Yaskawa INFORM job: A_ROOF_SIDE_0617_2_PAINT_11.JBI

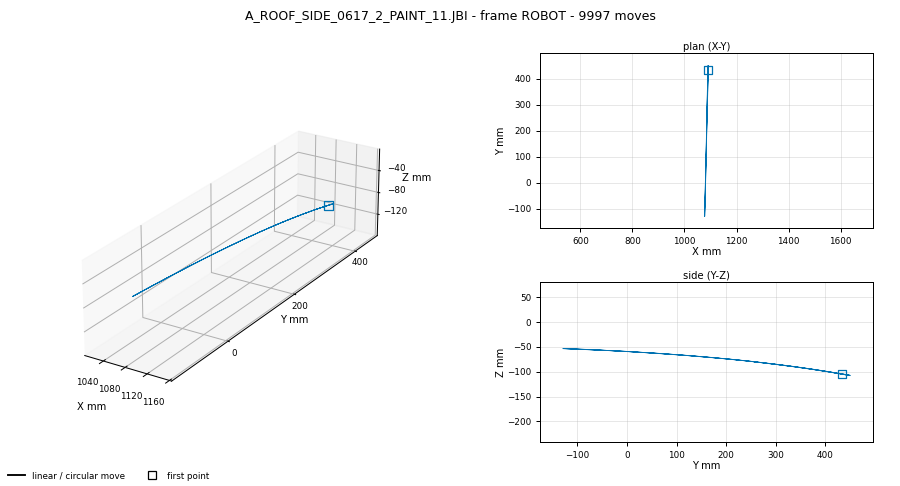
[picture p0: tool path of A_ROOF_SIDE_0617_2_PAINT_11.JBI in frame ROBOT, 9997 of 9997 moves have a stored position in this frame; points joined in program order, loops and branches not executed]
/JOB
//NAME A_ROOF_SIDE_0617_2_PAINT11
//POS
///NPOS 9997,0,0,0,0,0
///TOOL 1
///USER 0
///POSTYPE ROBOT
///RECTAN
///RCONF 1,0,0,0,0,0,0,0,0,0,0,0,0,0,0,0,0,0,0,0,0,0,0,0
C00000=1091.867,433.561,-104.062,178.470,26.056,154.096
C00001=1091.874,433.807,-104.105,178.473,26.068,154.099
C00002=1091.880,434.053,-104.148,178.477,26.080,154.102
C00003=1091.887,434.299,-104.192,178.480,26.092,154.104
C00004=1091.893,434.545,-104.234,178.484,26.104,154.107
C00005=1091.899,434.791,-104.277,178.486,26.116,154.110
C00006=1091.906,435.037,-104.321,178.490,26.128,154.112
C00007=1091.912,435.283,-104.365,178.493,26.141,154.115
C00008=1091.918,435.530,-104.408,178.497,26.153,154.117
C00009=1091.926,435.775,-104.451,178.500,26.165,154.120
C00010=1091.932,436.022,-104.494,178.503,26.177,154.123
C00011=1091.938,436.268,-104.538,178.507,26.189,154.126
C00012=1091.945,436.514,-104.581,178.510,26.202,154.128
C00013=1091.951,436.760,-104.624,178.513,26.214,154.131
C00014=1091.958,437.006,-104.668,178.517,26.227,154.134
C00015=1091.965,437.252,-104.711,178.520,26.239,154.137
C00016=1091.971,437.498,-104.755,178.524,26.252,154.139
C00017=1091.978,437.744,-104.799,178.527,26.264,154.142
C00018=1091.988,438.137,-104.869,178.533,26.285,154.147
C00019=1091.999,438.531,-104.938,178.538,26.305,154.151
C00020=1092.009,438.925,-105.008,178.543,26.326,154.156
C00021=1092.020,439.319,-105.078,178.548,26.346,154.160
C00022=1092.027,439.565,-105.122,178.552,26.359,154.163
C00023=1092.033,439.811,-105.166,178.556,26.372,154.166
C00024=1092.041,440.056,-105.210,178.559,26.385,154.169
C00025=1092.047,440.302,-105.254,178.562,26.398,154.172
C00026=1092.053,440.548,-105.297,178.565,26.411,154.175
C00027=1092.060,440.794,-105.341,178.569,26.424,154.178
C00028=1092.067,441.041,-105.385,178.572,26.438,154.181
C00029=1092.074,441.286,-105.430,178.575,26.451,154.184
C00030=1092.080,441.532,-105.474,178.579,26.464,154.187
C00031=1092.086,441.778,-105.518,178.583,26.478,154.190
C00032=1092.093,442.023,-105.562,178.586,26.491,154.193
C00033=1092.100,442.269,-105.606,178.589,26.504,154.196
C00034=1092.107,442.516,-105.650,178.593,26.518,154.199
C00035=1092.113,442.761,-105.695,178.596,26.532,154.202
C00036=1092.120,443.007,-105.739,178.600,26.546,154.205
C00037=1092.127,443.253,-105.783,178.603,26.559,154.208
C00038=1092.132,443.499,-105.828,178.606,26.573,154.211
C00039=1092.140,443.745,-105.873,178.610,26.586,154.214
C00040=1092.146,443.991,-105.917,178.614,26.601,154.218
C00041=1092.153,444.236,-105.961,178.616,26.614,154.221
C00042=1092.159,444.482,-106.006,178.620,26.628,154.224
C00043=1092.166,444.728,-106.050,178.624,26.642,154.227
C00044=1092.173,444.974,-106.094,178.626,26.656,154.230
C00045=1092.180,445.220,-106.140,178.629,26.670,154.233
C00046=1092.186,445.466,-106.185,178.632,26.684,154.237
C00047=1092.193,445.711,-106.228,178.633,26.697,154.240
C00048=1092.200,445.958,-106.273,178.636,26.711,154.243
C00049=1092.206,446.203,-106.318,178.638,26.725,154.246
C00050=1092.213,446.449,-106.363,178.639,26.739,154.250
C00051=1092.220,446.695,-106.408,178.641,26.752,154.253
C00052=1092.227,446.940,-106.453,178.643,26.767,154.256
C00053=1092.233,447.186,-106.498,178.644,26.780,154.260
C00054=1092.240,447.432,-106.543,178.645,26.794,154.263
C00055=1092.246,447.677,-106.588,178.646,26.807,154.267
C00056=1092.254,447.923,-106.633,178.647,26.821,154.270
C00057=1092.260,448.169,-106.677,178.648,26.835,154.273
C00058=1092.267,448.415,-106.723,178.648,26.849,154.277
C00059=1092.274,448.660,-106.767,178.649,26.862,154.280
C00060=1092.281,448.907,-106.812,178.649,26.876,154.284
C00061=1092.287,449.152,-106.857,178.650,26.890,154.287
C00062=1092.294,449.398,-106.902,178.649,26.903,154.291
C00063=1092.301,449.644,-106.947,178.649,26.917,154.294
C00064=1092.308,449.888,-106.992,178.649,26.931,154.298
C00065=1092.317,450.135,-107.036,178.649,26.943,154.301
C00066=1091.932,450.127,-107.217,178.601,27.145,154.357
C00067=1091.923,449.881,-107.173,178.601,27.132,154.354
C00068=1091.915,449.636,-107.127,178.601,27.119,154.350
C00069=1091.908,449.390,-107.082,178.601,27.105,154.347
C00070=1091.902,449.145,-107.037,178.601,27.091,154.343
C00071=1091.895,448.899,-106.992,178.601,27.078,154.340
C00072=1091.888,448.654,-106.947,178.601,27.064,154.336
C00073=1091.881,448.407,-106.902,178.600,27.050,154.333
C00074=1091.875,448.162,-106.857,178.600,27.037,154.330
C00075=1091.868,447.916,-106.811,178.599,27.023,154.326
C00076=1091.861,447.670,-106.767,178.598,27.009,154.323
C00077=1091.854,447.424,-106.722,178.596,26.995,154.319
C00078=1091.848,447.179,-106.677,178.595,26.982,154.316
C00079=1091.841,446.933,-106.632,178.594,26.968,154.313
C00080=1091.834,446.687,-106.587,178.592,26.954,154.309
C00081=1091.827,446.441,-106.542,178.591,26.940,154.306
C00082=1091.821,446.196,-106.497,178.588,26.926,154.303
C00083=1091.814,445.950,-106.453,178.586,26.912,154.299
C00084=1091.807,445.704,-106.407,178.585,26.898,154.296
C00085=1091.800,445.458,-106.363,178.582,26.884,154.293
C00086=1091.793,445.212,-106.318,178.579,26.871,154.290
C00087=1091.787,444.966,-106.274,178.576,26.857,154.286
C00088=1091.780,444.721,-106.229,178.573,26.843,154.283
C00089=1091.773,444.475,-106.184,178.570,26.829,154.280
C00090=1091.767,444.229,-106.139,178.567,26.815,154.277
C00091=1091.760,443.983,-106.095,178.563,26.801,154.274
C00092=1091.753,443.737,-106.050,178.559,26.787,154.270
C00093=1091.746,443.492,-106.006,178.556,26.773,154.267
C00094=1091.740,443.246,-105.962,178.553,26.760,154.264
C00095=1091.733,443.001,-105.917,178.549,26.746,154.261
C00096=1091.727,442.754,-105.873,178.545,26.732,154.258
C00097=1091.720,442.508,-105.828,178.542,26.718,154.255
C00098=1091.714,442.262,-105.784,178.539,26.705,154.252
C00099=1091.707,442.017,-105.740,178.535,26.691,154.249
C00100=1091.700,441.770,-105.695,178.531,26.678,154.246
C00101=1091.693,441.525,-105.651,178.527,26.664,154.243
C00102=1091.687,441.279,-105.607,178.525,26.651,154.240
C00103=1091.680,441.033,-105.563,178.521,26.637,154.237
C00104=1091.674,440.788,-105.519,178.517,26.624,154.234
C00105=1091.667,440.542,-105.475,178.514,26.611,154.231
C00106=1091.660,440.296,-105.431,178.510,26.598,154.228
C00107=1091.653,440.049,-105.387,178.508,26.585,154.225
C00108=1091.646,439.804,-105.343,178.504,26.572,154.222
C00109=1091.640,439.558,-105.299,178.500,26.559,154.219
C00110=1091.633,439.312,-105.255,178.497,26.546,154.216
C00111=1091.622,438.929,-105.187,178.491,26.526,154.212
C00112=1091.612,438.547,-105.119,178.486,26.506,154.207
C00113=1091.602,438.165,-105.050,178.481,26.486,154.203
C00114=1091.592,437.783,-104.983,178.475,26.466,154.198
C00115=1091.585,437.537,-104.939,178.471,26.454,154.196
C00116=1091.579,437.291,-104.896,178.469,26.441,154.193
C00117=1091.572,437.045,-104.853,178.465,26.428,154.190
C00118=1091.566,436.799,-104.809,178.462,26.416,154.187
C00119=1091.559,436.553,-104.765,178.458,26.403,154.185
C00120=1091.552,436.307,-104.722,178.455,26.391,154.182
C00121=1091.546,436.061,-104.678,178.451,26.378,154.179
C00122=1091.540,435.815,-104.635,178.448,26.367,154.176
C00123=1091.532,435.569,-104.591,178.444,26.354,154.174
C00124=1091.526,435.322,-104.548,178.441,26.342,154.171
C00125=1091.520,435.076,-104.504,178.437,26.329,154.168
C00126=1091.513,434.831,-104.461,178.434,26.317,154.166
C00127=1091.507,434.584,-104.418,178.431,26.305,154.163
C00128=1091.500,434.338,-104.374,178.427,26.293,154.160
C00129=1091.493,434.092,-104.332,178.424,26.281,154.158
C00130=1091.487,433.846,-104.288,178.420,26.268,154.155
C00131=1091.481,433.600,-104.246,178.417,26.257,154.152
C00132=1091.474,433.354,-104.202,178.414,26.245,154.150
C00133=1091.468,433.108,-104.159,178.410,26.233,154.147
C00134=1091.461,432.861,-104.116,178.407,26.221,154.144
C00135=1091.455,432.615,-104.072,178.403,26.209,154.142
C00136=1091.448,432.369,-104.030,178.400,26.197,154.139
C00137=1091.441,432.123,-103.987,178.397,26.186,154.137
C00138=1091.436,431.877,-103.944,178.393,26.174,154.134
C00139=1091.428,431.631,-103.901,178.390,26.162,154.132
C00140=1091.422,431.385,-103.858,178.387,26.151,154.129
C00141=1091.415,431.138,-103.815,178.383,26.139,154.127
C00142=1091.409,430.892,-103.773,178.380,26.128,154.124
C00143=1091.403,430.646,-103.730,178.377,26.117,154.122
C00144=1091.396,430.400,-103.688,178.374,26.105,154.119
C00145=1091.389,430.154,-103.645,178.370,26.094,154.117
C00146=1091.383,429.907,-103.602,178.367,26.082,154.114
C00147=1091.377,429.662,-103.560,178.364,26.071,154.112
C00148=1091.370,429.415,-103.517,178.360,26.060,154.110
C00149=1091.364,429.169,-103.474,178.356,26.048,154.107
C00150=1091.358,428.923,-103.432,178.353,26.037,154.105
C00151=1091.351,428.677,-103.389,178.350,26.026,154.102
C00152=1091.345,428.430,-103.346,178.347,26.015,154.100
C00153=1091.338,428.184,-103.304,178.343,26.004,154.097
C00154=1091.332,427.938,-103.261,178.340,25.993,154.095
C00155=1091.325,427.691,-103.220,178.337,25.982,154.093
C00156=1091.318,427.445,-103.177,178.333,25.971,154.090
C00157=1091.312,427.200,-103.135,178.330,25.960,154.088
C00158=1091.305,426.953,-103.092,178.326,25.949,154.086
C00159=1091.299,426.706,-103.050,178.323,25.938,154.083
C00160=1091.293,426.460,-103.008,178.320,25.927,154.081
C00161=1091.287,426.214,-102.966,178.317,25.916,154.079
C00162=1091.280,425.967,-102.923,178.313,25.906,154.077
C00163=1091.273,425.736,-102.884,178.310,25.895,154.074
C00164=1091.268,425.503,-102.844,178.307,25.885,154.072
C00165=1091.261,425.271,-102.804,178.304,25.876,154.070
C00166=1091.256,425.039,-102.765,178.301,25.866,154.068
C00167=1091.249,424.807,-102.725,178.298,25.856,154.066
C00168=1091.244,424.574,-102.686,178.294,25.846,154.064
C00169=1091.238,424.343,-102.646,178.292,25.836,154.062
C00170=1091.231,424.110,-102.607,178.288,25.826,154.060
C00171=1091.225,423.864,-102.565,178.285,25.815,154.057
C00172=1091.218,423.618,-102.523,178.282,25.805,154.055
C00173=1091.213,423.371,-102.481,178.279,25.794,154.053
C00174=1091.206,423.124,-102.440,178.275,25.784,154.051
C00175=1091.200,422.879,-102.397,178.272,25.774,154.049
C00176=1091.193,422.632,-102.356,178.269,25.764,154.046
C00177=1091.187,422.386,-102.314,178.266,25.753,154.044
C00178=1091.181,422.139,-102.272,178.262,25.743,154.042
C00179=1091.175,421.893,-102.231,178.259,25.733,154.040
C00180=1091.168,421.646,-102.188,178.256,25.723,154.038
C00181=1091.162,421.400,-102.147,178.252,25.713,154.036
C00182=1091.155,421.154,-102.106,178.249,25.703,154.034
C00183=1091.149,420.907,-102.064,178.246,25.693,154.032
C00184=1091.142,420.660,-102.022,178.243,25.682,154.029
C00185=1091.136,420.414,-101.981,178.239,25.672,154.027
C00186=1091.130,420.168,-101.939,178.236,25.662,154.025
C00187=1091.123,419.921,-101.898,178.233,25.653,154.023
C00188=1091.117,419.675,-101.857,178.229,25.642,154.021
C00189=1091.110,419.428,-101.815,178.226,25.633,154.019
C00190=1091.105,419.182,-101.773,178.223,25.623,154.017
C00191=1091.098,418.936,-101.733,178.219,25.613,154.015
C00192=1091.092,418.689,-101.691,178.217,25.603,154.013
C00193=1091.086,418.442,-101.650,178.214,25.594,154.011
C00194=1091.079,418.197,-101.609,178.210,25.584,154.009
C00195=1091.072,417.950,-101.567,178.207,25.574,154.007
C00196=1091.067,417.703,-101.527,178.204,25.564,154.005
C00197=1091.061,417.457,-101.485,178.200,25.555,154.003
C00198=1091.054,417.210,-101.444,178.197,25.545,154.001
C00199=1091.048,416.963,-101.403,178.194,25.536,153.999
C00200=1091.042,416.717,-101.362,178.191,25.526,153.997
C00201=1091.035,416.471,-101.321,178.187,25.517,153.995
C00202=1091.029,416.224,-101.280,178.184,25.507,153.993
C00203=1091.022,415.978,-101.239,178.181,25.497,153.991
C00204=1091.017,415.731,-101.198,178.177,25.488,153.989
C00205=1091.009,415.484,-101.157,178.175,25.479,153.987
C00206=1091.004,415.237,-101.116,178.171,25.470,153.985
C00207=1090.997,414.992,-101.075,178.168,25.461,153.984
C00208=1090.991,414.744,-101.034,178.165,25.451,153.982
C00209=1090.984,414.498,-100.994,178.162,25.442,153.980
C00210=1090.978,414.252,-100.953,178.159,25.433,153.978
C00211=1090.972,414.005,-100.912,178.155,25.424,153.976
C00212=1090.965,413.759,-100.872,178.152,25.414,153.974
C00213=1090.959,413.511,-100.830,178.149,25.405,153.972
C00214=1090.953,413.265,-100.790,178.146,25.396,153.970
C00215=1090.946,413.018,-100.750,178.142,25.387,153.969
C00216=1090.940,412.772,-100.709,178.140,25.378,153.967
C00217=1090.934,412.526,-100.669,178.136,25.369,153.965
C00218=1090.928,412.278,-100.627,178.133,25.360,153.963
C00219=1090.922,412.054,-100.591,178.130,25.352,153.961
C00220=1090.917,411.829,-100.554,178.127,25.344,153.960
C00221=1090.911,411.605,-100.517,178.124,25.336,153.958
C00222=1090.905,411.380,-100.480,178.122,25.328,153.957
C00223=1090.899,411.155,-100.443,178.119,25.319,153.955
C00224=1090.894,410.930,-100.406,178.115,25.311,153.953
C00225=1090.887,410.706,-100.370,178.112,25.303,153.952
C00226=1090.882,410.481,-100.333,178.110,25.295,153.950
C00227=1090.876,410.234,-100.293,178.107,25.287,153.948
C00228=1090.870,409.987,-100.252,178.103,25.278,153.947
C00229=1090.864,409.741,-100.212,178.100,25.269,153.945
C00230=1090.857,409.494,-100.171,178.097,25.260,153.943
C00231=1090.852,409.247,-100.131,178.094,25.252,153.941
C00232=1090.845,409.001,-100.091,178.091,25.243,153.939
C00233=1090.839,408.754,-100.051,178.088,25.234,153.938
C00234=1090.833,408.507,-100.011,178.084,25.226,153.936
C00235=1090.827,408.260,-99.970,178.082,25.217,153.934
C00236=1090.821,408.014,-99.930,178.078,25.208,153.933
C00237=1090.814,407.767,-99.890,178.075,25.200,153.931
C00238=1090.808,407.520,-99.851,178.072,25.192,153.929
C00239=1090.802,407.274,-99.810,178.069,25.183,153.927
C00240=1090.795,407.027,-99.770,178.065,25.175,153.926
C00241=1090.790,406.780,-99.729,178.063,25.166,153.924
C00242=1090.784,406.533,-99.690,178.059,25.158,153.923
C00243=1090.777,406.287,-99.650,178.057,25.149,153.921
C00244=1090.772,406.041,-99.610,178.053,25.141,153.919
C00245=1090.766,405.794,-99.571,178.050,25.133,153.918
C00246=1090.759,405.547,-99.531,178.047,25.124,153.916
C00247=1090.753,405.300,-99.491,178.044,25.116,153.914
C00248=1090.747,405.054,-99.451,178.040,25.108,153.913
C00249=1090.741,404.806,-99.412,178.038,25.100,153.911
C00250=1090.734,404.560,-99.371,178.035,25.092,153.909
C00251=1090.728,404.313,-99.332,178.031,25.084,153.908
C00252=1090.722,404.066,-99.292,178.029,25.076,153.906
C00253=1090.716,403.819,-99.252,178.025,25.067,153.905
C00254=1090.710,403.573,-99.213,178.022,25.059,153.903
C00255=1090.703,403.326,-99.174,178.018,25.051,153.902
C00256=1090.697,403.079,-99.134,178.016,25.043,153.900
C00257=1090.691,402.833,-99.094,178.013,25.035,153.898
C00258=1090.685,402.586,-99.055,178.009,25.027,153.897
C00259=1090.679,402.339,-99.015,178.007,25.019,153.895
C00260=1090.672,402.091,-98.976,178.004,25.011,153.894
C00261=1090.667,401.846,-98.936,178.000,25.003,153.892
C00262=1090.660,401.599,-98.897,177.997,24.996,153.891
C00263=1090.654,401.352,-98.858,177.994,24.988,153.889
C00264=1090.648,401.105,-98.818,177.991,24.980,153.888
C00265=1090.642,400.859,-98.779,177.988,24.972,153.886
C00266=1090.636,400.612,-98.739,177.984,24.964,153.885
C00267=1090.629,400.365,-98.700,177.982,24.956,153.883
C00268=1090.623,400.118,-98.661,177.979,24.949,153.882
C00269=1090.617,399.871,-98.622,177.975,24.941,153.880
C00270=1090.611,399.624,-98.582,177.972,24.933,153.878
C00271=1090.605,399.377,-98.543,177.970,24.925,153.877
C00272=1090.599,399.130,-98.504,177.967,24.918,153.876
C00273=1090.593,398.884,-98.465,177.963,24.910,153.874
C00274=1090.586,398.637,-98.426,177.960,24.903,153.873
C00275=1090.581,398.413,-98.390,177.957,24.896,153.871
C00276=1090.575,398.188,-98.355,177.954,24.889,153.870
C00277=1090.570,397.964,-98.320,177.952,24.882,153.869
C00278=1090.564,397.740,-98.283,177.949,24.875,153.867
C00279=1090.558,397.515,-98.249,177.946,24.868,153.866
C00280=1090.553,397.291,-98.213,177.943,24.862,153.865
C00281=1090.547,397.067,-98.177,177.941,24.855,153.863
C00282=1090.543,396.843,-98.142,177.938,24.848,153.862
C00283=1090.536,396.596,-98.103,177.935,24.841,153.861
C00284=1090.530,396.349,-98.064,177.931,24.833,153.859
C00285=1090.524,396.102,-98.026,177.929,24.826,153.858
C00286=1090.518,395.855,-97.987,177.926,24.818,153.857
C00287=1090.512,395.609,-97.948,177.923,24.811,153.855
C00288=1090.506,395.361,-97.910,177.919,24.803,153.854
C00289=1090.500,395.114,-97.870,177.916,24.796,153.852
C00290=1090.493,394.868,-97.832,177.913,24.789,153.851
C00291=1090.487,394.621,-97.793,177.910,24.782,153.850
C00292=1090.481,394.374,-97.755,177.907,24.774,153.848
C00293=1090.475,394.127,-97.716,177.904,24.767,153.847
C00294=1090.469,393.880,-97.677,177.901,24.760,153.846
C00295=1090.463,393.633,-97.639,177.898,24.753,153.844
C00296=1090.457,393.387,-97.601,177.895,24.746,153.843
C00297=1090.451,393.140,-97.561,177.892,24.738,153.841
C00298=1090.444,392.893,-97.523,177.889,24.731,153.840
C00299=1090.439,392.646,-97.484,177.885,24.724,153.839
C00300=1090.433,392.400,-97.446,177.882,24.717,153.838
C00301=1090.426,392.152,-97.408,177.879,24.710,153.836
C00302=1090.421,391.905,-97.369,177.876,24.703,153.835
C00303=1090.414,391.658,-97.330,177.873,24.696,153.834
C00304=1090.408,391.412,-97.293,177.870,24.689,153.832
C00305=1090.401,391.165,-97.254,177.866,24.682,153.831
C00306=1090.395,390.918,-97.216,177.864,24.675,153.830
C00307=1090.390,390.670,-97.177,177.860,24.668,153.829
C00308=1090.383,390.424,-97.139,177.858,24.661,153.827
C00309=1090.378,390.177,-97.101,177.855,24.654,153.826
C00310=1090.371,389.930,-97.063,177.852,24.648,153.825
C00311=1090.365,389.684,-97.025,177.849,24.641,153.823
C00312=1090.358,389.436,-96.986,177.846,24.634,153.822
C00313=1090.352,389.190,-96.949,177.842,24.627,153.821
C00314=1090.347,388.943,-96.910,177.839,24.620,153.820
C00315=1090.341,388.695,-96.872,177.836,24.613,153.819
C00316=1090.335,388.449,-96.834,177.833,24.606,153.817
C00317=1090.328,388.202,-96.796,177.830,24.600,153.816
C00318=1090.322,387.955,-96.758,177.827,24.593,153.815
C00319=1090.316,387.708,-96.720,177.824,24.586,153.813
C00320=1090.310,387.461,-96.682,177.821,24.580,153.812
C00321=1090.304,387.214,-96.644,177.818,24.573,153.811
C00322=1090.298,386.967,-96.606,177.815,24.566,153.810
C00323=1090.292,386.720,-96.569,177.812,24.559,153.809
C00324=1090.285,386.473,-96.531,177.807,24.553,153.808
C00325=1090.280,386.226,-96.492,177.804,24.546,153.806
C00326=1090.274,385.979,-96.454,177.801,24.539,153.805
C00327=1090.268,385.732,-96.417,177.798,24.533,153.804
C00328=1090.262,385.485,-96.379,177.795,24.526,153.803
C00329=1090.256,385.238,-96.341,177.792,24.520,153.802
C00330=1090.250,384.991,-96.303,177.789,24.513,153.800
C00331=1090.245,384.774,-96.270,177.787,24.507,153.799
C00332=1090.239,384.556,-96.236,177.784,24.502,153.798
C00333=1090.235,384.338,-96.203,177.781,24.496,153.797
C00334=1090.229,384.121,-96.171,177.779,24.490,153.796
C00335=1090.224,383.903,-96.137,177.776,24.485,153.795
C00336=1090.218,383.686,-96.104,177.774,24.479,153.794
C00337=1090.213,383.468,-96.070,177.770,24.473,153.793
C00338=1090.208,383.250,-96.038,177.768,24.467,153.792
C00339=1090.202,383.003,-96.000,177.765,24.461,153.791
C00340=1090.196,382.757,-95.963,177.762,24.454,153.790
C00341=1090.190,382.510,-95.925,177.759,24.448,153.789
C00342=1090.184,382.263,-95.888,177.756,24.442,153.788
C00343=1090.178,382.015,-95.850,177.752,24.435,153.786
C00344=1090.171,381.769,-95.812,177.749,24.429,153.785
C00345=1090.166,381.521,-95.775,177.746,24.423,153.784
C00346=1090.160,381.275,-95.738,177.743,24.416,153.783
C00347=1090.154,381.027,-95.701,177.740,24.410,153.782
C00348=1090.147,380.780,-95.663,177.737,24.404,153.781
C00349=1090.141,380.533,-95.626,177.734,24.397,153.780
C00350=1090.135,380.286,-95.588,177.731,24.391,153.779
C00351=1090.130,380.039,-95.551,177.727,24.385,153.778
C00352=1090.123,379.792,-95.514,177.724,24.379,153.777
C00353=1090.118,379.545,-95.477,177.721,24.373,153.776
C00354=1090.112,379.298,-95.439,177.718,24.367,153.774
C00355=1090.105,379.051,-95.403,177.716,24.361,153.773
C00356=1090.099,378.804,-95.365,177.713,24.355,153.772
C00357=1090.093,378.556,-95.328,177.709,24.348,153.771
C00358=1090.087,378.309,-95.291,177.706,24.342,153.770
C00359=1090.081,378.062,-95.254,177.703,24.336,153.769
C00360=1090.075,377.815,-95.216,177.700,24.330,153.768
C00361=1090.069,377.568,-95.180,177.697,24.324,153.767
C00362=1090.063,377.321,-95.142,177.694,24.318,153.766
C00363=1090.058,377.074,-95.105,177.690,24.312,153.765
C00364=1090.051,376.827,-95.069,177.687,24.306,153.764
C00365=1090.046,376.579,-95.032,177.684,24.300,153.763
C00366=1090.040,376.332,-94.995,177.682,24.294,153.762
C00367=1090.033,376.086,-94.958,177.679,24.288,153.761
C00368=1090.028,375.838,-94.921,177.675,24.282,153.760
C00369=1090.021,375.591,-94.884,177.672,24.276,153.759
C00370=1090.016,375.344,-94.847,177.669,24.270,153.758
C00371=1090.010,375.097,-94.810,177.666,24.264,153.757
C00372=1090.004,374.849,-94.774,177.663,24.258,153.756
C00373=1089.998,374.602,-94.737,177.660,24.252,153.755
C00374=1089.993,374.356,-94.700,177.657,24.246,153.754
C00375=1089.987,374.108,-94.663,177.654,24.240,153.753
C00376=1089.981,373.861,-94.627,177.651,24.235,153.752
C00377=1089.975,373.614,-94.590,177.647,24.229,153.751
C00378=1089.969,373.367,-94.553,177.644,24.223,153.750
C00379=1089.962,373.120,-94.517,177.641,24.217,153.749
C00380=1089.957,372.873,-94.480,177.639,24.212,153.748
C00381=1089.950,372.625,-94.444,177.635,24.206,153.747
C00382=1089.945,372.378,-94.406,177.632,24.200,153.746
C00383=1089.938,372.131,-94.370,177.629,24.194,153.745
C00384=1089.932,371.884,-94.334,177.626,24.188,153.744
C00385=1089.927,371.637,-94.297,177.623,24.183,153.743
C00386=1089.920,371.389,-94.261,177.620,24.177,153.742
C00387=1089.910,370.982,-94.200,177.615,24.168,153.741
C00388=1089.900,370.574,-94.141,177.610,24.158,153.739
C00389=1089.891,370.167,-94.081,177.605,24.149,153.738
C00390=1089.881,369.759,-94.021,177.599,24.140,153.736
C00391=1089.875,369.511,-93.984,177.596,24.134,153.735
C00392=1089.869,369.265,-93.948,177.594,24.129,153.734
C00393=1089.863,369.017,-93.912,177.590,24.123,153.733
C00394=1089.857,368.770,-93.876,177.587,24.118,153.732
C00395=1089.851,368.523,-93.839,177.584,24.112,153.731
C00396=1089.845,368.275,-93.803,177.580,24.106,153.731
C00397=1089.840,368.029,-93.767,177.578,24.101,153.730
C00398=1089.834,367.781,-93.731,177.575,24.095,153.729
C00399=1089.828,367.534,-93.694,177.571,24.090,153.728
C00400=1089.822,367.286,-93.658,177.568,24.084,153.727
C00401=1089.816,367.039,-93.622,177.566,24.079,153.726
C00402=1089.810,366.792,-93.586,177.563,24.073,153.725
C00403=1089.804,366.545,-93.550,177.559,24.068,153.724
C00404=1089.799,366.297,-93.514,177.556,24.062,153.723
C00405=1089.793,366.051,-93.478,177.553,24.057,153.722
C00406=1089.787,365.803,-93.442,177.550,24.052,153.722
C00407=1089.781,365.556,-93.406,177.547,24.046,153.721
C00408=1089.774,365.308,-93.370,177.544,24.041,153.720
C00409=1089.768,365.061,-93.334,177.541,24.035,153.719
C00410=1089.763,364.814,-93.299,177.538,24.030,153.718
C00411=1089.757,364.567,-93.262,177.534,24.025,153.717
C00412=1089.751,364.319,-93.226,177.532,24.019,153.716
C00413=1089.745,364.072,-93.191,177.529,24.014,153.716
C00414=1089.739,363.824,-93.155,177.525,24.008,153.715
C00415=1089.733,363.577,-93.119,177.523,24.003,153.714
C00416=1089.727,363.330,-93.083,177.519,23.998,153.713
C00417=1089.721,363.083,-93.048,177.516,23.993,153.712
C00418=1089.715,362.835,-93.012,177.513,23.987,153.711
C00419=1089.709,362.587,-92.976,177.510,23.982,153.711
C00420=1089.704,362.341,-92.940,177.507,23.977,153.710
C00421=1089.698,362.093,-92.905,177.503,23.971,153.709
C00422=1089.692,361.846,-92.869,177.501,23.967,153.708
C00423=1089.686,361.599,-92.833,177.498,23.961,153.707
C00424=1089.680,361.351,-92.798,177.494,23.956,153.706
C00425=1089.674,361.103,-92.762,177.492,23.951,153.706
C00426=1089.669,360.856,-92.727,177.488,23.946,153.705
C00427=1089.661,360.572,-92.686,177.485,23.940,153.704
C00428=1089.655,360.288,-92.645,177.481,23.934,153.703
C00429=1089.648,360.003,-92.604,177.478,23.928,153.702
C00430=1089.641,359.719,-92.564,177.474,23.922,153.701
C00431=1089.635,359.471,-92.528,177.471,23.917,153.700
C00432=1089.630,359.224,-92.493,177.468,23.912,153.700
C00433=1089.623,358.977,-92.457,177.465,23.907,153.699
C00434=1089.617,358.729,-92.422,177.462,23.902,153.698
C00435=1089.612,358.482,-92.386,177.458,23.897,153.697
C00436=1089.606,358.234,-92.351,177.456,23.892,153.697
C00437=1089.600,357.987,-92.317,177.453,23.886,153.696
C00438=1089.594,357.739,-92.281,177.450,23.882,153.695
C00439=1089.585,357.384,-92.230,177.445,23.875,153.694
C00440=1089.577,357.029,-92.179,177.440,23.867,153.693
C00441=1089.568,356.674,-92.129,177.437,23.860,153.692
C00442=1089.560,356.319,-92.078,177.432,23.853,153.691
C00443=1089.553,356.072,-92.043,177.428,23.848,153.690
C00444=1089.548,355.825,-92.008,177.426,23.843,153.689
C00445=1089.542,355.577,-91.973,177.422,23.838,153.688
C00446=1089.536,355.330,-91.938,177.420,23.833,153.688
C00447=1089.530,355.082,-91.903,177.416,23.828,153.687
C00448=1089.525,354.835,-91.868,177.413,23.823,153.686
C00449=1089.519,354.588,-91.833,177.410,23.818,153.685
C00450=1089.513,354.340,-91.798,177.407,23.813,153.685
C00451=1089.508,354.093,-91.763,177.404,23.809,153.684
C00452=1089.501,353.845,-91.728,177.401,23.804,153.683
C00453=1089.496,353.598,-91.693,177.398,23.799,153.682
C00454=1089.489,353.350,-91.658,177.395,23.794,153.682
C00455=1089.484,353.103,-91.623,177.391,23.789,153.681
C00456=1089.478,352.854,-91.588,177.389,23.784,153.680
C00457=1089.472,352.608,-91.553,177.385,23.779,153.680
C00458=1089.466,352.360,-91.518,177.383,23.775,153.679
C00459=1089.460,352.112,-91.484,177.379,23.770,153.678
C00460=1089.454,351.865,-91.449,177.377,23.765,153.678
C00461=1089.448,351.617,-91.414,177.373,23.761,153.677
C00462=1089.442,351.371,-91.380,177.371,23.756,153.676
C00463=1089.437,351.122,-91.345,177.367,23.751,153.676
C00464=1089.431,350.875,-91.311,177.364,23.746,153.675
C00465=1089.425,350.627,-91.276,177.361,23.742,153.674
C00466=1089.419,350.380,-91.241,177.357,23.737,153.673
C00467=1089.414,350.132,-91.206,177.355,23.732,153.673
C00468=1089.407,349.885,-91.172,177.351,23.727,153.672
C00469=1089.401,349.638,-91.137,177.349,23.723,153.671
C00470=1089.395,349.390,-91.102,177.345,23.718,153.671
C00471=1089.390,349.142,-91.068,177.343,23.714,153.670
C00472=1089.384,348.895,-91.033,177.339,23.709,153.669
C00473=1089.378,348.647,-90.999,177.337,23.704,153.669
C00474=1089.372,348.399,-90.965,177.333,23.699,153.668
C00475=1089.367,348.152,-90.930,177.330,23.695,153.667
C00476=1089.360,347.904,-90.895,177.327,23.690,153.667
C00477=1089.354,347.657,-90.861,177.324,23.685,153.666
C00478=1089.349,347.410,-90.826,177.321,23.681,153.665
C00479=1089.343,347.162,-90.792,177.318,23.676,153.665
C00480=1089.337,346.914,-90.758,177.315,23.671,153.664
C00481=1089.332,346.667,-90.723,177.312,23.667,153.663
C00482=1089.326,346.419,-90.689,177.308,23.662,153.663
C00483=1089.319,346.171,-90.655,177.306,23.658,153.662
C00484=1089.314,345.924,-90.620,177.302,23.653,153.661
C00485=1089.308,345.677,-90.586,177.300,23.649,153.661
C00486=1089.302,345.429,-90.552,177.296,23.644,153.660
C00487=1089.296,345.181,-90.518,177.293,23.639,153.659
C00488=1089.291,344.934,-90.483,177.290,23.635,153.659
C00489=1089.285,344.686,-90.450,177.287,23.630,153.658
C00490=1089.279,344.438,-90.415,177.284,23.626,153.658
C00491=1089.270,344.049,-90.362,177.279,23.619,153.657
C00492=1089.261,343.660,-90.308,177.274,23.612,153.656
C00493=1089.251,343.270,-90.254,177.269,23.605,153.655
C00494=1089.242,342.881,-90.201,177.265,23.598,153.654
C00495=1089.236,342.633,-90.167,177.262,23.594,153.653
C00496=1089.231,342.386,-90.133,177.259,23.589,153.652
C00497=1089.225,342.138,-90.099,177.255,23.585,153.652
C00498=1089.218,341.890,-90.065,177.253,23.581,153.651
C00499=1089.213,341.643,-90.031,177.249,23.576,153.651
C00500=1089.207,341.395,-89.997,177.246,23.571,153.650
C00501=1089.201,341.148,-89.963,177.243,23.567,153.650
C00502=1089.195,340.900,-89.930,177.240,23.563,153.649
C00503=1089.189,340.652,-89.895,177.237,23.558,153.648
C00504=1089.183,340.404,-89.862,177.234,23.554,153.648
C00505=1089.178,340.157,-89.828,177.231,23.550,153.647
C00506=1089.172,339.909,-89.795,177.228,23.545,153.647
C00507=1089.166,339.662,-89.761,177.225,23.541,153.646
C00508=1089.160,339.414,-89.727,177.222,23.537,153.645
C00509=1089.155,339.166,-89.693,177.219,23.532,153.645
C00510=1089.149,338.919,-89.659,177.216,23.528,153.644
C00511=1089.143,338.671,-89.626,177.212,23.523,153.644
C00512=1089.137,338.423,-89.592,177.210,23.519,153.643
C00513=1089.131,338.175,-89.558,177.207,23.515,153.643
C00514=1089.126,337.927,-89.525,177.203,23.511,153.642
C00515=1089.120,337.680,-89.491,177.200,23.507,153.641
C00516=1089.114,337.432,-89.457,177.198,23.503,153.641
C00517=1089.108,337.185,-89.423,177.194,23.498,153.640
C00518=1089.102,336.937,-89.391,177.191,23.494,153.640
C00519=1089.097,336.690,-89.357,177.188,23.489,153.639
C00520=1089.091,336.442,-89.323,177.185,23.485,153.639
C00521=1089.085,336.194,-89.290,177.182,23.481,153.638
C00522=1089.079,335.946,-89.256,177.179,23.477,153.637
C00523=1089.073,335.698,-89.223,177.176,23.473,153.637
C00524=1089.067,335.451,-89.189,177.173,23.468,153.636
C00525=1089.061,335.203,-89.156,177.170,23.464,153.636
C00526=1089.056,334.955,-89.123,177.167,23.460,153.635
C00527=1089.050,334.707,-89.089,177.164,23.456,153.635
C00528=1089.044,334.460,-89.056,177.160,23.452,153.634
C00529=1089.038,334.212,-89.023,177.158,23.448,153.634
C00530=1089.033,333.964,-88.989,177.155,23.444,153.633
C00531=1089.027,333.716,-88.956,177.151,23.439,153.633
C00532=1089.021,333.469,-88.923,177.149,23.435,153.632
C00533=1089.015,333.221,-88.890,177.146,23.431,153.631
C00534=1089.010,332.973,-88.856,177.142,23.427,153.631
C00535=1089.004,332.725,-88.823,177.139,23.423,153.630
C00536=1088.997,332.478,-88.790,177.137,23.419,153.630
C00537=1088.992,332.230,-88.756,177.133,23.414,153.629
C00538=1088.986,331.982,-88.723,177.130,23.410,153.629
C00539=1088.980,331.735,-88.690,177.128,23.406,153.628
C00540=1088.974,331.487,-88.657,177.124,23.402,153.628
C00541=1088.968,331.239,-88.624,177.121,23.398,153.627
C00542=1088.963,330.991,-88.591,177.118,23.394,153.627
C00543=1088.953,330.596,-88.539,177.113,23.388,153.626
C00544=1088.944,330.201,-88.486,177.108,23.382,153.625
C00545=1088.935,329.806,-88.434,177.103,23.375,153.624
C00546=1088.925,329.411,-88.381,177.098,23.369,153.624
C00547=1088.919,329.164,-88.348,177.095,23.365,153.623
C00548=1088.914,328.915,-88.316,177.092,23.361,153.623
C00549=1088.907,328.667,-88.283,177.090,23.357,153.622
C00550=1088.901,328.420,-88.250,177.086,23.353,153.622
C00551=1088.896,328.172,-88.217,177.083,23.349,153.621
C00552=1088.889,327.924,-88.184,177.080,23.345,153.621
C00553=1088.884,327.676,-88.152,177.077,23.341,153.620
C00554=1088.878,327.428,-88.119,177.074,23.337,153.620
C00555=1088.871,327.181,-88.086,177.071,23.334,153.619
C00556=1088.867,326.933,-88.054,177.068,23.329,153.619
C00557=1088.860,326.685,-88.021,177.065,23.325,153.618
C00558=1088.854,326.438,-87.988,177.062,23.322,153.618
C00559=1088.849,326.189,-87.956,177.059,23.318,153.617
C00560=1088.843,325.942,-87.923,177.056,23.314,153.617
C00561=1088.837,325.694,-87.890,177.052,23.310,153.617
C00562=1088.831,325.445,-87.858,177.050,23.306,153.616
C00563=1088.825,325.199,-87.825,177.047,23.302,153.616
C00564=1088.819,324.951,-87.793,177.044,23.299,153.615
C00565=1088.814,324.702,-87.760,177.040,23.294,153.615
C00566=1088.808,324.455,-87.727,177.037,23.290,153.614
C00567=1088.802,324.207,-87.695,177.035,23.287,153.614
C00568=1088.797,323.959,-87.662,177.032,23.283,153.613
C00569=1088.791,323.711,-87.630,177.029,23.279,153.613
C00570=1088.784,323.464,-87.597,177.025,23.275,153.612
C00571=1088.779,323.215,-87.565,177.022,23.271,153.612
C00572=1088.773,322.968,-87.532,177.020,23.268,153.611
C00573=1088.767,322.720,-87.500,177.017,23.264,153.611
C00574=1088.761,322.472,-87.468,177.014,23.260,153.610
C00575=1088.756,322.225,-87.435,177.010,23.256,153.610
C00576=1088.750,321.976,-87.403,177.007,23.252,153.610
C00577=1088.744,321.729,-87.371,177.004,23.248,153.609
C00578=1088.738,321.481,-87.339,177.002,23.245,153.609
C00579=1088.734,321.233,-87.306,176.998,23.240,153.608
C00580=1088.727,320.985,-87.274,176.995,23.237,153.608
C00581=1088.721,320.737,-87.242,176.992,23.233,153.607
C00582=1088.716,320.489,-87.210,176.989,23.229,153.607
C00583=1088.710,320.241,-87.177,176.987,23.226,153.606
C00584=1088.704,319.993,-87.145,176.984,23.222,153.606
C00585=1088.699,319.746,-87.113,176.980,23.217,153.605
C00586=1088.693,319.498,-87.081,176.977,23.214,153.605
C00587=1088.687,319.251,-87.048,176.974,23.210,153.605
C00588=1088.682,319.002,-87.016,176.972,23.206,153.604
C00589=1088.676,318.754,-86.984,176.969,23.203,153.604
C00590=1088.671,318.506,-86.952,176.965,23.199,153.603
C00591=1088.665,318.258,-86.920,176.962,23.195,153.603
C00592=1088.659,318.011,-86.888,176.959,23.191,153.602
C00593=1088.653,317.763,-86.856,176.956,23.188,153.602
C00594=1088.648,317.515,-86.823,176.954,23.184,153.602
C00595=1088.639,317.113,-86.771,176.949,23.178,153.601
C00596=1088.630,316.711,-86.720,176.944,23.171,153.600
C00597=1088.621,316.309,-86.668,176.939,23.166,153.599
C00598=1088.612,315.907,-86.616,176.934,23.159,153.599
C00599=1088.606,315.659,-86.585,176.931,23.156,153.598
C00600=1088.600,315.411,-86.553,176.929,23.152,153.598
C00601=1088.595,315.163,-86.521,176.925,23.148,153.597
C00602=1088.589,314.915,-86.489,176.922,23.144,153.597
C00603=1088.583,314.667,-86.457,176.919,23.141,153.597
C00604=1088.577,314.420,-86.426,176.916,23.138,153.596
C00605=1088.571,314.171,-86.394,176.913,23.134,153.596
C00606=1088.565,313.924,-86.362,176.910,23.131,153.595
C00607=1088.559,313.676,-86.330,176.907,23.127,153.595
C00608=1088.553,313.428,-86.299,176.904,23.123,153.595
C00609=1088.547,313.180,-86.267,176.901,23.120,153.594
C00610=1088.541,312.932,-86.235,176.898,23.116,153.594
C00611=1088.536,312.684,-86.204,176.895,23.112,153.593
C00612=1088.530,312.436,-86.173,176.892,23.109,153.593
C00613=1088.524,312.189,-86.141,176.889,23.106,153.593
C00614=1088.518,311.940,-86.109,176.886,23.102,153.592
C00615=1088.512,311.693,-86.078,176.883,23.099,153.592
C00616=1088.506,311.444,-86.047,176.879,23.095,153.592
C00617=1088.501,311.197,-86.015,176.876,23.091,153.591
C00618=1088.494,310.949,-85.983,176.873,23.088,153.591
C00619=1088.489,310.701,-85.952,176.871,23.084,153.590
C00620=1088.483,310.453,-85.921,176.868,23.081,153.590
C00621=1088.478,310.205,-85.889,176.865,23.077,153.590
C00622=1088.471,309.957,-85.857,176.862,23.074,153.589
C00623=1088.466,309.709,-85.826,176.859,23.070,153.589
C00624=1088.459,309.461,-85.795,176.856,23.067,153.589
C00625=1088.454,309.213,-85.764,176.853,23.064,153.588
C00626=1088.449,308.965,-85.732,176.849,23.059,153.588
C00627=1088.442,308.718,-85.701,176.846,23.056,153.588
C00628=1088.437,308.469,-85.670,176.843,23.053,153.587
C00629=1088.431,308.221,-85.638,176.841,23.049,153.587
C00630=1088.425,307.973,-85.608,176.838,23.046,153.586
C00631=1088.420,307.726,-85.576,176.835,23.042,153.586
C00632=1088.413,307.477,-85.545,176.832,23.039,153.586
C00633=1088.408,307.230,-85.514,176.829,23.035,153.585
C00634=1088.403,306.982,-85.483,176.826,23.032,153.585
C00635=1088.396,306.734,-85.451,176.823,23.028,153.584
C00636=1088.391,306.486,-85.420,176.820,23.025,153.584
C00637=1088.385,306.238,-85.389,176.816,23.021,153.584
C00638=1088.379,305.990,-85.358,176.813,23.018,153.583
C00639=1088.373,305.742,-85.327,176.810,23.014,153.583
C00640=1088.368,305.494,-85.296,176.807,23.011,153.583
C00641=1088.361,305.246,-85.264,176.805,23.007,153.582
C00642=1088.356,304.998,-85.234,176.802,23.004,153.582
C00643=1088.351,304.750,-85.203,176.799,23.000,153.582
C00644=1088.345,304.503,-85.172,176.796,22.997,153.581
C00645=1088.339,304.254,-85.140,176.793,22.994,153.581
C00646=1088.334,304.006,-85.110,176.790,22.990,153.581
C00647=1088.324,303.607,-85.060,176.785,22.984,153.580
C00648=1088.315,303.208,-85.010,176.780,22.979,153.579
C00649=1088.306,302.808,-84.960,176.775,22.973,153.579
C00650=1088.298,302.410,-84.910,176.771,22.968,153.578
C00651=1088.291,302.161,-84.880,176.768,22.965,153.578
C00652=1088.286,301.913,-84.849,176.765,22.961,153.577
C00653=1088.280,301.665,-84.818,176.762,22.958,153.577
C00654=1088.275,301.418,-84.787,176.759,22.954,153.577
C00655=1088.269,301.170,-84.756,176.755,22.950,153.576
C00656=1088.264,300.922,-84.726,176.752,22.947,153.576
C00657=1088.257,300.673,-84.695,176.749,22.944,153.576
C00658=1088.252,300.426,-84.664,176.746,22.940,153.575
C00659=1088.247,300.177,-84.634,176.744,22.937,153.575
C00660=1088.241,299.930,-84.603,176.741,22.934,153.575
C00661=1088.236,299.681,-84.572,176.738,22.930,153.574
C00662=1088.230,299.434,-84.542,176.735,22.927,153.574
C00663=1088.225,299.185,-84.511,176.732,22.923,153.574
C00664=1088.219,298.938,-84.481,176.729,22.920,153.573
C00665=1088.213,298.689,-84.450,176.726,22.917,153.573
C00666=1088.207,298.441,-84.419,176.723,22.913,153.573
C00667=1088.202,298.193,-84.389,176.720,22.910,153.572
C00668=1088.196,297.945,-84.358,176.717,22.906,153.572
C00669=1088.191,297.697,-84.327,176.714,22.903,153.572
C00670=1088.185,297.449,-84.297,176.711,22.900,153.571
C00671=1088.179,297.202,-84.267,176.708,22.896,153.571
C00672=1088.173,296.954,-84.236,176.705,22.893,153.571
C00673=1088.167,296.705,-84.205,176.702,22.889,153.570
C00674=1088.162,296.456,-84.175,176.699,22.886,153.570
C00675=1088.156,296.209,-84.145,176.696,22.883,153.570
C00676=1088.150,295.961,-84.115,176.693,22.880,153.569
C00677=1088.145,295.713,-84.084,176.690,22.877,153.569
C00678=1088.139,295.465,-84.054,176.687,22.873,153.569
C00679=1088.133,295.217,-84.023,176.684,22.870,153.568
C00680=1088.128,294.969,-83.994,176.681,22.866,153.568
C00681=1088.122,294.721,-83.964,176.678,22.863,153.568
C00682=1088.116,294.473,-83.933,176.675,22.860,153.568
C00683=1088.110,294.224,-83.902,176.672,22.857,153.567
C00684=1088.105,293.976,-83.872,176.669,22.854,153.567
C00685=1088.099,293.728,-83.842,176.666,22.850,153.567
C00686=1088.093,293.480,-83.812,176.664,22.847,153.566
C00687=1088.088,293.232,-83.782,176.661,22.844,153.566
C00688=1088.082,292.984,-83.752,176.659,22.841,153.566
C00689=1088.076,292.736,-83.721,176.656,22.838,153.565
C00690=1088.070,292.488,-83.692,176.653,22.834,153.565
C00691=1088.065,292.240,-83.661,176.650,22.831,153.565
C00692=1088.059,291.992,-83.632,176.647,22.828,153.564
C00693=1088.053,291.744,-83.601,176.644,22.825,153.564
C00694=1088.047,291.496,-83.571,176.641,22.821,153.564
C00695=1088.042,291.247,-83.541,176.638,22.818,153.564
C00696=1088.036,291.000,-83.511,176.635,22.815,153.563
C00697=1088.031,290.751,-83.481,176.632,22.812,153.563
C00698=1088.025,290.503,-83.451,176.629,22.808,153.563
C00699=1088.016,290.119,-83.405,176.624,22.804,153.562
C00700=1088.007,289.733,-83.359,176.620,22.799,153.562
C00701=1087.999,289.348,-83.312,176.615,22.793,153.561
C00702=1087.989,288.962,-83.266,176.611,22.789,153.561
C00703=1087.983,288.714,-83.236,176.608,22.786,153.561
C00704=1087.978,288.466,-83.206,176.605,22.782,153.560
C00705=1087.972,288.218,-83.176,176.602,22.779,153.560
C00706=1087.966,287.970,-83.147,176.599,22.776,153.560
C00707=1087.960,287.722,-83.117,176.596,22.773,153.559
C00708=1087.954,287.474,-83.087,176.593,22.770,153.559
C00709=1087.949,287.225,-83.057,176.590,22.766,153.559
C00710=1087.944,286.978,-83.028,176.587,22.763,153.558
C00711=1087.937,286.730,-82.998,176.584,22.760,153.558
C00712=1087.932,286.482,-82.969,176.581,22.757,153.558
C00713=1087.926,286.233,-82.939,176.578,22.753,153.558
C00714=1087.921,285.985,-82.909,176.575,22.751,153.557
C00715=1087.915,285.737,-82.880,176.572,22.748,153.557
C00716=1087.909,285.489,-82.850,176.570,22.745,153.557
C00717=1087.903,285.240,-82.820,176.567,22.741,153.557
C00718=1087.898,284.992,-82.791,176.564,22.738,153.556
C00719=1087.891,284.744,-82.762,176.561,22.735,153.556
C00720=1087.887,284.496,-82.732,176.558,22.732,153.556
C00721=1087.881,284.248,-82.702,176.555,22.729,153.555
C00722=1087.875,284.000,-82.673,176.552,22.725,153.555
C00723=1087.869,283.752,-82.643,176.549,22.722,153.555
C00724=1087.863,283.503,-82.614,176.546,22.719,153.555
C00725=1087.858,283.255,-82.584,176.543,22.717,153.554
C00726=1087.852,283.007,-82.555,176.540,22.713,153.554
C00727=1087.847,282.759,-82.526,176.537,22.710,153.554
C00728=1087.841,282.510,-82.496,176.534,22.707,153.554
C00729=1087.835,282.262,-82.467,176.531,22.704,153.553
C00730=1087.830,282.014,-82.437,176.528,22.701,153.553
C00731=1087.825,281.766,-82.408,176.525,22.697,153.553
C00732=1087.818,281.518,-82.379,176.522,22.694,153.552
C00733=1087.813,281.270,-82.350,176.520,22.691,153.552
C00734=1087.807,281.021,-82.320,176.517,22.688,153.552
C00735=1087.801,280.773,-82.291,176.514,22.685,153.552
C00736=1087.795,280.526,-82.262,176.511,22.682,153.551
C00737=1087.790,280.277,-82.233,176.508,22.679,153.551
C00738=1087.784,280.029,-82.204,176.505,22.676,153.551
C00739=1087.779,279.780,-82.175,176.502,22.673,153.551
C00740=1087.772,279.532,-82.146,176.499,22.670,153.550
C00741=1087.767,279.284,-82.116,176.497,22.667,153.550
C00742=1087.761,279.036,-82.087,176.494,22.664,153.550
C00743=1087.756,278.787,-82.058,176.491,22.661,153.550
C00744=1087.749,278.539,-82.029,176.488,22.658,153.549
C00745=1087.745,278.291,-82.000,176.485,22.654,153.549
C00746=1087.738,278.043,-81.971,176.482,22.651,153.549
C00747=1087.733,277.794,-81.941,176.480,22.648,153.548
C00748=1087.727,277.547,-81.913,176.476,22.646,153.548
C00749=1087.722,277.298,-81.884,176.474,22.642,153.548
C00750=1087.716,277.050,-81.855,176.471,22.639,153.548
C00751=1087.707,276.674,-81.811,176.466,22.635,153.547
C00752=1087.699,276.299,-81.767,176.461,22.630,153.547
C00753=1087.690,275.923,-81.723,176.458,22.626,153.547
C00754=1087.682,275.547,-81.680,176.453,22.621,153.546
C00755=1087.676,275.299,-81.650,176.450,22.618,153.546
C00756=1087.670,275.050,-81.622,176.447,22.615,153.546
C00757=1087.664,274.803,-81.593,176.444,22.612,153.545
C00758=1087.659,274.554,-81.564,176.441,22.609,153.545
C00759=1087.653,274.306,-81.535,176.439,22.606,153.545
C00760=1087.647,274.058,-81.507,176.436,22.603,153.545
C00761=1087.642,273.809,-81.478,176.433,22.600,153.544
C00762=1087.636,273.561,-81.449,176.430,22.597,153.544
C00763=1087.631,273.313,-81.421,176.427,22.594,153.544
C00764=1087.624,273.065,-81.392,176.424,22.591,153.544
C00765=1087.620,272.816,-81.363,176.422,22.588,153.543
C00766=1087.614,272.568,-81.335,176.419,22.585,153.543
C00767=1087.607,272.320,-81.306,176.415,22.582,153.543
C00768=1087.602,272.072,-81.278,176.412,22.579,153.543
C00769=1087.597,271.823,-81.248,176.409,22.576,153.542
C00770=1087.591,271.574,-81.220,176.407,22.573,153.542
C00771=1087.585,271.327,-81.191,176.404,22.570,153.542
C00772=1087.579,271.078,-81.163,176.401,22.567,153.542
C00773=1087.574,270.830,-81.135,176.398,22.564,153.542
C00774=1087.567,270.582,-81.106,176.395,22.561,153.541
C00775=1087.562,270.333,-81.077,176.393,22.558,153.541
C00776=1087.557,270.085,-81.049,176.390,22.555,153.541
C00777=1087.551,269.837,-81.020,176.387,22.552,153.540
C00778=1087.545,269.589,-80.992,176.384,22.549,153.540
C00779=1087.539,269.340,-80.964,176.381,22.546,153.540
C00780=1087.534,269.092,-80.936,176.378,22.544,153.540
C00781=1087.528,268.844,-80.907,176.375,22.540,153.540
C00782=1087.522,268.595,-80.878,176.373,22.537,153.539
C00783=1087.517,268.347,-80.850,176.369,22.534,153.539
C00784=1087.511,268.098,-80.822,176.366,22.531,153.539
C00785=1087.506,267.850,-80.793,176.364,22.529,153.539
C00786=1087.500,267.602,-80.764,176.361,22.526,153.538
C00787=1087.494,267.354,-80.736,176.358,22.523,153.538
C00788=1087.488,267.105,-80.708,176.355,22.520,153.538
C00789=1087.483,266.857,-80.680,176.353,22.517,153.538
C00790=1087.477,266.608,-80.652,176.350,22.514,153.538
C00791=1087.472,266.360,-80.624,176.347,22.511,153.537
C00792=1087.466,266.112,-80.595,176.344,22.508,153.537
C00793=1087.460,265.864,-80.567,176.341,22.505,153.537
C00794=1087.454,265.615,-80.538,176.338,22.502,153.537
C00795=1087.449,265.367,-80.511,176.335,22.499,153.536
C00796=1087.443,265.118,-80.482,176.332,22.496,153.536
C00797=1087.438,264.870,-80.454,176.329,22.493,153.536
C00798=1087.432,264.622,-80.426,176.327,22.490,153.536
C00799=1087.426,264.373,-80.398,176.324,22.488,153.535
C00800=1087.420,264.125,-80.370,176.321,22.484,153.535
C00801=1087.414,263.877,-80.342,176.318,22.482,153.535
C00802=1087.408,263.628,-80.314,176.316,22.479,153.535
C00803=1087.400,263.255,-80.273,176.311,22.475,153.535
C00804=1087.392,262.882,-80.230,176.307,22.470,153.534
C00805=1087.383,262.510,-80.188,176.303,22.466,153.534
C00806=1087.374,262.138,-80.146,176.298,22.462,153.534
C00807=1087.368,261.888,-80.119,176.295,22.459,153.533
C00808=1087.362,261.640,-80.091,176.293,22.456,153.533
C00809=1087.356,261.392,-80.063,176.290,22.453,153.533
C00810=1087.351,261.144,-80.035,176.287,22.450,153.533
C00811=1087.345,260.895,-80.007,176.284,22.447,153.533
C00812=1087.339,260.647,-79.979,176.281,22.445,153.532
C00813=1087.333,260.398,-79.952,176.278,22.442,153.532
C00814=1087.328,260.150,-79.924,176.275,22.439,153.532
C00815=1087.322,259.902,-79.897,176.273,22.436,153.532
C00816=1087.316,259.653,-79.868,176.270,22.434,153.531
C00817=1087.311,259.405,-79.841,176.267,22.431,153.531
C00818=1087.304,259.156,-79.813,176.264,22.428,153.531
C00819=1087.299,258.908,-79.785,176.262,22.425,153.531
C00820=1087.294,258.659,-79.758,176.259,22.422,153.531
C00821=1087.287,258.411,-79.730,176.256,22.419,153.530
C00822=1087.282,258.163,-79.702,176.253,22.416,153.530
C00823=1087.277,257.914,-79.675,176.250,22.414,153.530
C00824=1087.270,257.666,-79.647,176.247,22.411,153.530
C00825=1087.265,257.418,-79.619,176.244,22.408,153.530
C00826=1087.259,257.169,-79.592,176.242,22.405,153.529
C00827=1087.253,256.921,-79.564,176.239,22.402,153.529
C00828=1087.248,256.672,-79.537,176.236,22.399,153.529
C00829=1087.242,256.424,-79.510,176.233,22.396,153.529
C00830=1087.236,256.175,-79.482,176.231,22.394,153.529
C00831=1087.231,255.927,-79.454,176.227,22.391,153.528
C00832=1087.225,255.679,-79.427,176.224,22.388,153.528
C00833=1087.219,255.430,-79.399,176.222,22.385,153.528
C00834=1087.213,255.182,-79.372,176.219,22.382,153.528
C00835=1087.208,254.933,-79.345,176.216,22.379,153.528
C00836=1087.202,254.684,-79.318,176.214,22.377,153.527
C00837=1087.197,254.436,-79.290,176.211,22.374,153.527
C00838=1087.192,254.187,-79.262,176.208,22.371,153.527
C00839=1087.185,253.940,-79.235,176.206,22.368,153.527
C00840=1087.180,253.690,-79.207,176.202,22.365,153.526
C00841=1087.174,253.443,-79.180,176.200,22.362,153.526
C00842=1087.169,253.194,-79.153,176.196,22.359,153.526
C00843=1087.163,252.946,-79.126,176.194,22.357,153.526
C00844=1087.158,252.698,-79.098,176.191,22.354,153.526
C00845=1087.151,252.448,-79.071,176.188,22.351,153.525
C00846=1087.146,252.200,-79.044,176.186,22.348,153.525
C00847=1087.141,251.952,-79.016,176.183,22.345,153.525
C00848=1087.135,251.703,-78.989,176.180,22.342,153.525
C00849=1087.130,251.455,-78.962,176.178,22.340,153.525
C00850=1087.123,251.206,-78.934,176.175,22.337,153.524
C00851=1087.118,250.958,-78.907,176.171,22.334,153.524
C00852=1087.113,250.709,-78.881,176.169,22.331,153.524
C00853=1087.107,250.461,-78.853,176.166,22.328,153.524
C00854=1087.101,250.213,-78.826,176.163,22.325,153.524
C00855=1087.093,249.837,-78.785,176.159,22.321,153.523
C00856=1087.085,249.461,-78.744,176.155,22.317,153.523
C00857=1087.076,249.085,-78.703,176.151,22.313,153.523
C00858=1087.068,248.710,-78.663,176.147,22.308,153.522
C00859=1087.063,248.461,-78.635,176.144,22.305,153.522
C00860=1087.057,248.213,-78.609,176.141,22.303,153.522
C00861=1087.052,247.964,-78.581,176.138,22.299,153.521
C00862=1087.046,247.716,-78.554,176.136,22.297,153.521
C00863=1087.040,247.468,-78.527,176.133,22.294,153.521
C00864=1087.035,247.219,-78.500,176.130,22.291,153.521
C00865=1087.029,246.970,-78.473,176.128,22.289,153.521
C00866=1087.023,246.722,-78.446,176.125,22.285,153.520
C00867=1087.018,246.473,-78.419,176.122,22.283,153.520
C00868=1087.012,246.225,-78.393,176.119,22.280,153.520
C00869=1087.006,245.976,-78.366,176.116,22.277,153.520
C00870=1087.001,245.728,-78.339,176.113,22.274,153.520
C00871=1086.996,245.479,-78.312,176.111,22.272,153.520
C00872=1086.990,245.231,-78.285,176.108,22.269,153.519
C00873=1086.984,244.983,-78.259,176.106,22.266,153.519
C00874=1086.978,244.734,-78.232,176.103,22.263,153.519
C00875=1086.973,244.485,-78.206,176.100,22.260,153.519
C00876=1086.968,244.237,-78.179,176.097,22.258,153.519
C00877=1086.962,243.988,-78.152,176.095,22.255,153.518
C00878=1086.956,243.739,-78.125,176.091,22.252,153.518
C00879=1086.951,243.490,-78.098,176.089,22.250,153.518
C00880=1086.945,243.242,-78.071,176.086,22.246,153.518
C00881=1086.939,242.994,-78.045,176.084,22.244,153.517
C00882=1086.933,242.745,-78.019,176.081,22.241,153.517
C00883=1086.928,242.496,-77.992,176.078,22.238,153.517
C00884=1086.922,242.248,-77.965,176.076,22.236,153.517
C00885=1086.916,242.000,-77.939,176.072,22.233,153.517
C00886=1086.910,241.751,-77.912,176.069,22.230,153.517
C00887=1086.905,241.502,-77.886,176.067,22.227,153.516
C00888=1086.899,241.254,-77.860,176.064,22.224,153.516
C00889=1086.893,241.006,-77.833,176.062,22.222,153.516
C00890=1086.888,240.757,-77.806,176.059,22.219,153.516
C00891=1086.883,240.508,-77.780,176.056,22.216,153.516
C00892=1086.877,240.260,-77.753,176.054,22.214,153.515
C00893=1086.871,240.011,-77.726,176.050,22.211,153.515
C00894=1086.866,239.762,-77.701,176.048,22.208,153.515
C00895=1086.860,239.514,-77.674,176.045,22.205,153.515
C00896=1086.854,239.266,-77.648,176.042,22.202,153.515
C00897=1086.848,239.017,-77.622,176.040,22.200,153.514
C00898=1086.842,238.769,-77.595,176.037,22.197,153.514
C00899=1086.837,238.520,-77.569,176.035,22.195,153.514
C00900=1086.831,238.271,-77.543,176.031,22.192,153.514
C00901=1086.825,238.023,-77.516,176.029,22.188,153.514
C00902=1086.820,237.774,-77.490,176.026,22.186,153.514
C00903=1086.814,237.525,-77.463,176.023,22.183,153.513
C00904=1086.809,237.277,-77.438,176.021,22.181,153.513
C00905=1086.803,237.029,-77.411,176.018,22.178,153.513
C00906=1086.798,236.780,-77.385,176.016,22.175,153.513
C00907=1086.788,236.397,-77.345,176.011,22.171,153.512
C00908=1086.781,236.014,-77.304,176.007,22.167,153.512
C00909=1086.772,235.632,-77.264,176.003,22.162,153.512
C00910=1086.763,235.250,-77.224,175.999,22.159,153.512
C00911=1086.757,235.001,-77.198,175.996,22.155,153.511
C00912=1086.752,234.753,-77.172,175.993,22.153,153.511
C00913=1086.746,234.504,-77.146,175.991,22.150,153.511
C00914=1086.741,234.255,-77.120,175.988,22.147,153.511
C00915=1086.736,234.007,-77.093,175.985,22.145,153.511
C00916=1086.730,233.758,-77.068,175.982,22.142,153.510
C00917=1086.724,233.510,-77.042,175.980,22.139,153.510
C00918=1086.718,233.261,-77.016,175.977,22.136,153.510
C00919=1086.713,233.012,-76.990,175.975,22.134,153.510
C00920=1086.707,232.763,-76.964,175.972,22.131,153.510
C00921=1086.701,232.515,-76.938,175.969,22.128,153.510
C00922=1086.696,232.267,-76.912,175.967,22.125,153.509
C00923=1086.690,232.018,-76.886,175.963,22.123,153.509
C00924=1086.685,231.769,-76.860,175.961,22.120,153.509
C00925=1086.678,231.521,-76.834,175.958,22.117,153.509
C00926=1086.673,231.272,-76.808,175.956,22.115,153.509
C00927=1086.668,231.023,-76.783,175.953,22.112,153.508
C00928=1086.663,230.774,-76.757,175.951,22.110,153.508
C00929=1086.656,230.526,-76.731,175.948,22.106,153.508
C00930=1086.651,230.277,-76.705,175.945,22.104,153.508
C00931=1086.645,230.028,-76.679,175.942,22.101,153.508
C00932=1086.640,229.780,-76.654,175.939,22.098,153.508
C00933=1086.634,229.531,-76.628,175.937,22.096,153.507
C00934=1086.628,229.283,-76.603,175.934,22.093,153.507
C00935=1086.622,229.034,-76.577,175.932,22.090,153.507
C00936=1086.617,228.785,-76.551,175.929,22.088,153.507
C00937=1086.611,228.537,-76.525,175.926,22.085,153.507
C00938=1086.606,228.288,-76.499,175.923,22.082,153.507
C00939=1086.599,228.040,-76.474,175.921,22.080,153.506
C00940=1086.594,227.791,-76.448,175.918,22.077,153.506
C00941=1086.588,227.543,-76.423,175.916,22.074,153.506
C00942=1086.583,227.294,-76.397,175.913,22.072,153.506
C00943=1086.577,227.045,-76.372,175.911,22.069,153.505
C00944=1086.571,226.796,-76.346,175.908,22.066,153.505
C00945=1086.566,226.548,-76.321,175.905,22.064,153.505
C00946=1086.560,226.299,-76.295,175.902,22.061,153.505
C00947=1086.554,226.051,-76.269,175.900,22.059,153.505
C00948=1086.549,225.802,-76.244,175.897,22.055,153.505
C00949=1086.543,225.554,-76.219,175.895,22.053,153.504
C00950=1086.538,225.304,-76.193,175.892,22.050,153.504
C00951=1086.531,225.055,-76.168,175.889,22.048,153.504
C00952=1086.527,224.807,-76.142,175.886,22.044,153.504
C00953=1086.520,224.558,-76.117,175.884,22.042,153.504
C00954=1086.515,224.309,-76.091,175.881,22.039,153.504
C00955=1086.509,224.062,-76.066,175.879,22.037,153.503
C00956=1086.504,223.813,-76.040,175.876,22.034,153.503
C00957=1086.498,223.565,-76.015,175.874,22.031,153.503
C00958=1086.493,223.315,-75.990,175.871,22.029,153.503
C00959=1086.484,222.924,-75.951,175.867,22.024,153.502
C00960=1086.475,222.533,-75.910,175.862,22.020,153.502
C00961=1086.466,222.142,-75.870,175.859,22.016,153.502
C00962=1086.457,221.751,-75.831,175.854,22.012,153.502
C00963=1086.452,221.502,-75.805,175.852,22.009,153.501
C00964=1086.446,221.254,-75.780,175.849,22.006,153.501
C00965=1086.440,221.004,-75.756,175.847,22.004,153.501
C00966=1086.435,220.755,-75.730,175.843,22.001,153.501
C00967=1086.429,220.507,-75.705,175.841,21.999,153.501
C00968=1086.423,220.258,-75.680,175.838,21.996,153.501
C00969=1086.418,220.010,-75.655,175.836,21.993,153.500
C00970=1086.412,219.761,-75.629,175.833,21.990,153.500
C00971=1086.406,219.512,-75.605,175.831,21.988,153.500
C00972=1086.401,219.264,-75.580,175.828,21.985,153.500
C00973=1086.395,219.015,-75.554,175.825,21.983,153.500
C00974=1086.390,218.766,-75.529,175.823,21.980,153.499
C00975=1086.384,218.518,-75.504,175.820,21.977,153.499
C00976=1086.378,218.268,-75.480,175.818,21.975,153.499
C00977=1086.372,218.020,-75.455,175.815,21.972,153.499
C00978=1086.366,217.771,-75.430,175.812,21.969,153.499
C00979=1086.362,217.523,-75.404,175.810,21.966,153.499
C00980=1086.355,217.274,-75.379,175.807,21.964,153.498
C00981=1086.350,217.026,-75.355,175.804,21.961,153.498
C00982=1086.344,216.776,-75.330,175.802,21.959,153.498
C00983=1086.339,216.528,-75.305,175.800,21.956,153.498
C00984=1086.333,216.279,-75.280,175.797,21.953,153.498
C00985=1086.328,216.031,-75.255,175.795,21.951,153.498
C00986=1086.322,215.782,-75.230,175.791,21.948,153.497
C00987=1086.316,215.534,-75.205,175.789,21.945,153.497
C00988=1086.310,215.284,-75.181,175.786,21.942,153.497
C00989=1086.305,215.036,-75.156,175.784,21.940,153.497
C00990=1086.300,214.787,-75.131,175.781,21.937,153.497
C00991=1086.294,214.538,-75.106,175.779,21.935,153.497
C00992=1086.288,214.289,-75.081,175.776,21.932,153.496
C00993=1086.283,214.041,-75.057,175.774,21.929,153.496
C00994=1086.278,213.792,-75.032,175.771,21.927,153.496
C00995=1086.271,213.544,-75.007,175.768,21.924,153.496
C00996=1086.266,213.295,-74.983,175.766,21.922,153.496
C00997=1086.260,213.046,-74.958,175.763,21.918,153.495
C00998=1086.255,212.798,-74.933,175.761,21.916,153.495
C00999=1086.249,212.548,-74.909,175.759,21.913,153.495
C01000=1086.243,212.300,-74.884,175.755,21.911,153.495
C01001=1086.237,212.051,-74.860,175.753,21.908,153.495
C01002=1086.232,211.803,-74.835,175.750,21.905,153.495
C01003=1086.227,211.554,-74.811,175.748,21.903,153.494
C01004=1086.221,211.305,-74.786,175.745,21.900,153.494
C01005=1086.215,211.056,-74.762,175.743,21.898,153.494
C01006=1086.209,210.807,-74.736,175.740,21.895,153.494
C01007=1086.204,210.559,-74.712,175.738,21.892,153.494
C01008=1086.199,210.310,-74.688,175.735,21.889,153.493
C01009=1086.193,210.061,-74.663,175.732,21.887,153.493
C01010=1086.187,209.812,-74.639,175.730,21.884,153.493
C01011=1086.179,209.425,-74.600,175.726,21.880,153.493
C01012=1086.170,209.038,-74.563,175.722,21.876,153.493
C01013=1086.160,208.651,-74.525,175.718,21.872,153.492
C01014=1086.153,208.264,-74.486,175.714,21.868,153.492
C01015=1086.130,207.237,-74.388,175.634,21.826,153.495
C01016=1086.123,206.988,-74.364,175.631,21.824,153.495
C01017=1086.118,206.739,-74.340,175.629,21.823,153.496
C01018=1086.112,206.490,-74.315,175.626,21.821,153.496
C01019=1086.107,206.241,-74.292,175.624,21.819,153.495
C01020=1086.101,205.993,-74.268,175.620,21.817,153.496
C01021=1086.095,205.744,-74.244,175.618,21.816,153.496
C01022=1086.090,205.495,-74.221,175.615,21.814,153.496
C01023=1086.084,205.246,-74.196,175.613,21.812,153.496
C01024=1086.078,204.998,-74.173,175.610,21.811,153.496
C01025=1086.073,204.749,-74.149,175.608,21.809,153.496
C01026=1086.068,204.500,-74.125,175.604,21.807,153.496
C01027=1086.062,204.250,-74.102,175.602,21.805,153.496
C01028=1086.056,204.002,-74.077,175.599,21.804,153.496
C01029=1086.050,203.754,-74.054,175.597,21.802,153.496
C01030=1086.045,203.504,-74.030,175.594,21.800,153.496
C01031=1086.040,203.256,-74.006,175.592,21.798,153.496
C01032=1086.034,203.007,-73.983,175.589,21.797,153.496
C01033=1086.029,202.758,-73.959,175.586,21.795,153.496
C01034=1086.023,202.509,-73.936,175.583,21.793,153.496
C01035=1086.017,202.260,-73.911,175.581,21.792,153.496
C01036=1086.012,202.011,-73.888,175.578,21.790,153.496
C01037=1086.006,201.763,-73.864,175.576,21.788,153.496
C01038=1086.001,201.514,-73.841,175.573,21.787,153.496
C01039=1085.995,201.265,-73.817,175.571,21.785,153.496
C01040=1085.990,201.016,-73.794,175.568,21.784,153.496
C01041=1085.984,200.768,-73.770,175.565,21.781,153.496
C01042=1085.977,200.518,-73.747,175.562,21.780,153.497
C01043=1085.972,200.270,-73.723,175.560,21.778,153.497
C01044=1085.966,200.021,-73.700,175.557,21.777,153.497
C01045=1085.960,199.773,-73.676,175.555,21.775,153.497
C01046=1085.955,199.523,-73.652,175.552,21.773,153.497
C01047=1085.950,199.275,-73.629,175.550,21.772,153.497
C01048=1085.944,199.026,-73.606,175.547,21.770,153.497
C01049=1085.939,198.777,-73.582,175.544,21.768,153.497
C01050=1085.933,198.528,-73.559,175.541,21.766,153.497
C01051=1085.927,198.280,-73.536,175.539,21.765,153.497
C01052=1085.922,198.031,-73.512,175.536,21.763,153.497
C01053=1085.915,197.781,-73.489,175.533,21.762,153.497
C01054=1085.909,197.533,-73.465,175.531,21.760,153.497
C01055=1085.904,197.284,-73.442,175.528,21.758,153.497
C01056=1085.899,197.035,-73.419,175.526,21.757,153.497
C01057=1085.893,196.786,-73.395,175.524,21.755,153.497
C01058=1085.887,196.538,-73.372,175.521,21.753,153.497
C01059=1085.882,196.288,-73.348,175.518,21.751,153.497
C01060=1085.876,196.039,-73.326,175.515,21.750,153.497
C01061=1085.870,195.791,-73.303,175.513,21.748,153.497
C01062=1085.865,195.542,-73.278,175.510,21.746,153.497
C01063=1085.859,195.293,-73.255,175.507,21.745,153.497
C01064=1085.854,195.044,-73.232,175.505,21.743,153.497
C01065=1085.848,194.795,-73.209,175.502,21.741,153.498
C01066=1085.843,194.546,-73.186,175.500,21.740,153.497
C01067=1085.837,194.298,-73.162,175.497,21.738,153.498
C01068=1085.831,194.049,-73.139,175.495,21.736,153.498
C01069=1085.825,193.800,-73.116,175.493,21.734,153.498
C01070=1085.820,193.551,-73.093,175.490,21.733,153.498
C01071=1085.815,193.302,-73.070,175.487,21.731,153.498
C01072=1085.809,193.053,-73.047,175.484,21.729,153.498
C01073=1085.804,192.805,-73.024,175.482,21.728,153.498
C01074=1085.799,192.556,-73.001,175.479,21.726,153.498
C01075=1085.793,192.307,-72.977,175.476,21.724,153.498
C01076=1085.787,192.029,-72.952,175.474,21.722,153.498
C01077=1085.780,191.750,-72.926,175.471,21.720,153.498
C01078=1085.774,191.472,-72.900,175.468,21.718,153.498
C01079=1085.768,191.194,-72.874,175.466,21.717,153.498
C01080=1085.762,190.945,-72.851,175.463,21.715,153.498
C01081=1085.757,190.697,-72.829,175.461,21.713,153.498
C01082=1085.752,190.448,-72.805,175.457,21.711,153.498
C01083=1085.746,190.199,-72.782,175.455,21.710,153.498
C01084=1085.740,189.950,-72.759,175.452,21.708,153.498
C01085=1085.735,189.701,-72.736,175.450,21.706,153.498
C01086=1085.729,189.452,-72.713,175.447,21.704,153.498
C01087=1085.724,189.203,-72.690,175.445,21.703,153.498
C01088=1085.718,188.954,-72.667,175.443,21.701,153.498
C01089=1085.713,188.706,-72.645,175.440,21.699,153.498
C01090=1085.708,188.457,-72.622,175.437,21.697,153.498
C01091=1085.702,188.208,-72.599,175.435,21.696,153.498
C01092=1085.696,187.959,-72.576,175.432,21.694,153.498
C01093=1085.690,187.710,-72.553,175.430,21.692,153.498
C01094=1085.686,187.461,-72.530,175.428,21.691,153.498
C01095=1085.680,187.213,-72.507,175.425,21.689,153.498
C01096=1085.675,186.964,-72.484,175.423,21.687,153.498
C01097=1085.669,186.714,-72.462,175.420,21.685,153.498
C01098=1085.663,186.465,-72.439,175.418,21.684,153.498
C01099=1085.658,186.217,-72.416,175.415,21.682,153.498
C01100=1085.653,185.968,-72.394,175.413,21.680,153.498
C01101=1085.647,185.719,-72.371,175.410,21.678,153.498
C01102=1085.642,185.469,-72.348,175.408,21.677,153.498
C01103=1085.637,185.221,-72.325,175.405,21.675,153.498
C01104=1085.631,184.972,-72.302,175.403,21.673,153.498
C01105=1085.625,184.724,-72.280,175.400,21.671,153.498
C01106=1085.619,184.474,-72.258,175.398,21.670,153.499
C01107=1085.614,184.225,-72.235,175.395,21.668,153.499
C01108=1085.608,183.976,-72.212,175.393,21.667,153.499
C01109=1085.602,183.727,-72.190,175.390,21.665,153.499
C01110=1085.597,183.479,-72.168,175.388,21.664,153.499
C01111=1085.591,183.230,-72.145,175.385,21.662,153.499
C01112=1085.585,182.981,-72.122,175.383,21.660,153.499
C01113=1085.580,182.732,-72.099,175.380,21.659,153.499
C01114=1085.573,182.483,-72.077,175.378,21.657,153.499
C01115=1085.568,182.234,-72.055,175.375,21.655,153.499
C01116=1085.562,181.985,-72.032,175.373,21.653,153.499
C01117=1085.556,181.737,-72.010,175.370,21.652,153.499
C01118=1085.551,181.487,-71.988,175.368,21.650,153.499
C01119=1085.545,181.238,-71.965,175.365,21.648,153.499
C01120=1085.540,180.989,-71.942,175.362,21.647,153.499
C01121=1085.533,180.740,-71.920,175.360,21.645,153.499
C01122=1085.528,180.492,-71.898,175.357,21.644,153.499
C01123=1085.523,180.243,-71.875,175.355,21.642,153.499
C01124=1085.516,179.994,-71.853,175.353,21.640,153.499
C01125=1085.511,179.744,-71.831,175.350,21.639,153.499
C01126=1085.506,179.496,-71.808,175.348,21.637,153.499
C01127=1085.499,179.247,-71.787,175.345,21.635,153.499
C01128=1085.494,178.998,-71.764,175.342,21.634,153.499
C01129=1085.488,178.749,-71.741,175.340,21.632,153.499
C01130=1085.483,178.500,-71.719,175.337,21.630,153.500
C01131=1085.477,178.251,-71.697,175.335,21.629,153.500
C01132=1085.471,178.002,-71.674,175.333,21.627,153.499
C01133=1085.466,177.753,-71.652,175.331,21.626,153.500
C01134=1085.460,177.504,-71.631,175.328,21.624,153.500
C01135=1085.455,177.255,-71.608,175.326,21.622,153.500
C01136=1085.448,177.006,-71.586,175.323,21.621,153.500
C01137=1085.443,176.757,-71.563,175.321,21.619,153.500
C01138=1085.438,176.509,-71.541,175.319,21.617,153.500
C01139=1085.432,176.259,-71.520,175.316,21.616,153.500
C01140=1085.425,175.981,-71.495,175.313,21.614,153.500
C01141=1085.419,175.703,-71.470,175.310,21.611,153.500
C01142=1085.413,175.424,-71.445,175.308,21.609,153.500
C01143=1085.406,175.146,-71.420,175.305,21.608,153.500
C01144=1085.401,174.896,-71.398,175.303,21.606,153.500
C01145=1085.396,174.648,-71.376,175.300,21.604,153.500
C01146=1085.390,174.399,-71.354,175.298,21.603,153.500
C01147=1085.384,174.149,-71.332,175.295,21.601,153.500
C01148=1085.378,173.901,-71.310,175.293,21.599,153.500
C01149=1085.373,173.652,-71.288,175.290,21.597,153.500
C01150=1085.368,173.403,-71.266,175.288,21.596,153.500
C01151=1085.362,173.154,-71.244,175.285,21.594,153.500
C01152=1085.356,172.905,-71.221,175.283,21.592,153.500
C01153=1085.351,172.657,-71.200,175.280,21.590,153.500
C01154=1085.345,172.407,-71.178,175.279,21.589,153.500
C01155=1085.341,172.158,-71.156,175.277,21.587,153.500
C01156=1085.334,171.910,-71.133,175.274,21.586,153.500
C01157=1085.329,171.660,-71.111,175.271,21.584,153.500
C01158=1085.323,171.412,-71.090,175.269,21.582,153.500
C01159=1085.318,171.162,-71.068,175.267,21.580,153.500
C01160=1085.312,170.914,-71.046,175.264,21.578,153.500
C01161=1085.307,170.664,-71.024,175.262,21.577,153.500
C01162=1085.301,170.416,-71.003,175.259,21.575,153.500
C01163=1085.295,170.167,-70.980,175.257,21.573,153.500
C01164=1085.289,169.917,-70.958,175.254,21.571,153.500
C01165=1085.284,169.669,-70.936,175.253,21.570,153.500
C01166=1085.279,169.419,-70.914,175.250,21.569,153.500
C01167=1085.273,169.171,-70.893,175.248,21.567,153.500
C01168=1085.268,168.921,-70.871,175.245,21.565,153.500
C01169=1085.262,168.673,-70.849,175.243,21.563,153.500
C01170=1085.257,168.423,-70.827,175.240,21.561,153.500
C01171=1085.251,168.175,-70.806,175.238,21.559,153.500
C01172=1085.246,167.925,-70.784,175.236,21.557,153.500
C01173=1085.240,167.677,-70.762,175.233,21.556,153.500
C01174=1085.235,167.427,-70.740,175.231,21.555,153.500
C01175=1085.229,167.179,-70.719,175.229,21.553,153.500
C01176=1085.224,166.929,-70.697,175.227,21.551,153.500
C01177=1085.218,166.681,-70.675,175.224,21.549,153.500
C01178=1085.212,166.431,-70.654,175.222,21.547,153.500
C01179=1085.207,166.183,-70.632,175.219,21.545,153.500
C01180=1085.202,165.934,-70.611,175.217,21.543,153.500
C01181=1085.196,165.684,-70.588,175.214,21.541,153.500
C01182=1085.191,165.436,-70.567,175.213,21.541,153.500
C01183=1085.186,165.186,-70.545,175.210,21.539,153.500
C01184=1085.180,164.938,-70.524,175.208,21.537,153.500
C01185=1085.175,164.688,-70.501,175.205,21.535,153.500
C01186=1085.169,164.440,-70.480,175.203,21.533,153.500
C01187=1085.164,164.191,-70.459,175.201,21.531,153.500
C01188=1085.158,163.941,-70.437,175.198,21.529,153.500
C01189=1085.153,163.693,-70.416,175.196,21.527,153.500
C01190=1085.147,163.443,-70.394,175.194,21.526,153.500
C01191=1085.142,163.195,-70.373,175.192,21.524,153.500
C01192=1085.137,162.946,-70.351,175.189,21.522,153.500
C01193=1085.131,162.696,-70.330,175.187,21.520,153.500
C01194=1085.126,162.447,-70.308,175.185,21.519,153.500
C01195=1085.121,162.199,-70.287,175.182,21.517,153.500
C01196=1085.114,161.950,-70.265,175.180,21.515,153.500
C01197=1085.110,161.701,-70.243,175.178,21.513,153.500
C01198=1085.104,161.451,-70.222,175.176,21.512,153.500
C01199=1085.098,161.202,-70.201,175.173,21.510,153.500
C01200=1085.093,160.954,-70.180,175.171,21.508,153.500
C01201=1085.087,160.704,-70.158,175.168,21.506,153.500
C01202=1085.082,160.455,-70.137,175.166,21.505,153.500
C01203=1085.076,160.206,-70.115,175.164,21.503,153.500
C01204=1085.069,159.927,-70.092,175.161,21.501,153.500
C01205=1085.063,159.648,-70.068,175.159,21.499,153.500
C01206=1085.057,159.369,-70.044,175.156,21.497,153.500
C01207=1085.051,159.091,-70.021,175.154,21.495,153.500
C01208=1085.045,158.842,-69.999,175.151,21.493,153.500
C01209=1085.040,158.593,-69.978,175.149,21.491,153.500
C01210=1085.034,158.344,-69.956,175.147,21.490,153.500
C01211=1085.029,158.095,-69.935,175.145,21.489,153.500
C01212=1085.023,157.846,-69.914,175.142,21.487,153.500
C01213=1085.017,157.597,-69.893,175.140,21.485,153.500
C01214=1085.012,157.348,-69.872,175.137,21.483,153.500
C01215=1085.006,157.099,-69.851,175.135,21.481,153.500
C01216=1085.000,156.850,-69.829,175.133,21.479,153.500
C01217=1084.995,156.601,-69.809,175.131,21.478,153.500
C01218=1084.989,156.352,-69.787,175.129,21.476,153.500
C01219=1084.984,156.102,-69.766,175.126,21.474,153.500
C01220=1084.978,155.854,-69.745,175.124,21.472,153.500
C01221=1084.973,155.605,-69.724,175.121,21.470,153.500
C01222=1084.967,155.355,-69.702,175.120,21.469,153.500
C01223=1084.962,155.106,-69.682,175.117,21.467,153.500
C01224=1084.957,154.858,-69.661,175.115,21.465,153.500
C01225=1084.951,154.608,-69.640,175.112,21.464,153.500
C01226=1084.944,154.360,-69.619,175.110,21.462,153.500
C01227=1084.939,154.111,-69.598,175.108,21.461,153.500
C01228=1084.933,153.861,-69.577,175.106,21.459,153.500
C01229=1084.928,153.612,-69.556,175.104,21.457,153.500
C01230=1084.922,153.364,-69.535,175.101,21.455,153.500
C01231=1084.916,153.114,-69.514,175.099,21.453,153.500
C01232=1084.911,152.865,-69.494,175.097,21.452,153.500
C01233=1084.905,152.616,-69.472,175.095,21.450,153.500
C01234=1084.900,152.366,-69.451,175.092,21.448,153.500
C01235=1084.894,152.118,-69.430,175.090,21.446,153.500
C01236=1084.889,151.869,-69.410,175.088,21.444,153.500
C01237=1084.884,151.620,-69.389,175.086,21.443,153.499
C01238=1084.877,151.370,-69.367,175.084,21.441,153.499
C01239=1084.872,151.121,-69.347,175.081,21.439,153.499
C01240=1084.867,150.872,-69.326,175.079,21.437,153.499
C01241=1084.861,150.624,-69.305,175.077,21.436,153.499
C01242=1084.855,150.374,-69.284,175.075,21.434,153.499
C01243=1084.849,150.125,-69.264,175.072,21.432,153.499
C01244=1084.844,149.877,-69.243,175.070,21.430,153.499
C01245=1084.839,149.627,-69.222,175.068,21.428,153.499
C01246=1084.833,149.378,-69.201,175.066,21.427,153.499
C01247=1084.827,149.129,-69.180,175.064,21.425,153.499
C01248=1084.822,148.880,-69.160,175.061,21.423,153.499
C01249=1084.817,148.631,-69.139,175.059,21.421,153.499
C01250=1084.811,148.382,-69.119,175.057,21.420,153.499
C01251=1084.805,148.132,-69.098,175.055,21.418,153.499
C01252=1084.799,147.884,-69.077,175.052,21.416,153.499
C01253=1084.794,147.635,-69.056,175.050,21.414,153.499
C01254=1084.789,147.385,-69.036,175.048,21.413,153.499
C01255=1084.782,147.136,-69.015,175.046,21.411,153.499
C01256=1084.777,146.887,-68.995,175.044,21.409,153.499
C01257=1084.771,146.638,-68.974,175.041,21.407,153.499
C01258=1084.765,146.390,-68.954,175.040,21.406,153.499
C01259=1084.759,146.140,-68.933,175.037,21.404,153.499
C01260=1084.754,145.891,-68.912,175.035,21.402,153.499
C01261=1084.749,145.641,-68.892,175.032,21.400,153.499
C01262=1084.743,145.393,-68.872,175.031,21.399,153.499
C01263=1084.738,145.144,-68.851,175.028,21.397,153.499
C01264=1084.732,144.895,-68.830,175.026,21.395,153.499
C01265=1084.726,144.645,-68.809,175.024,21.393,153.499
C01266=1084.720,144.396,-68.789,175.022,21.391,153.499
C01267=1084.715,144.147,-68.768,175.020,21.390,153.499
C01268=1084.709,143.868,-68.746,175.017,21.387,153.499
C01269=1084.703,143.589,-68.723,175.015,21.385,153.499
C01270=1084.696,143.311,-68.700,175.013,21.383,153.499
C01271=1084.690,143.031,-68.677,175.010,21.382,153.499
C01272=1084.684,142.782,-68.656,175.008,21.380,153.499
C01273=1084.679,142.533,-68.636,175.005,21.378,153.499
C01274=1084.673,142.284,-68.616,175.003,21.375,153.499
C01275=1084.668,142.035,-68.595,175.002,21.374,153.498
C01276=1084.662,141.785,-68.574,174.999,21.372,153.498
C01277=1084.656,141.536,-68.554,174.997,21.370,153.498
C01278=1084.651,141.287,-68.534,174.994,21.368,153.498
C01279=1084.645,141.039,-68.514,174.993,21.367,153.498
C01280=1084.640,140.789,-68.493,174.990,21.365,153.498
C01281=1084.635,140.540,-68.473,174.988,21.363,153.498
C01282=1084.629,140.291,-68.454,174.986,21.361,153.498
C01283=1084.623,140.042,-68.433,174.984,21.359,153.498
C01284=1084.617,139.793,-68.413,174.982,21.357,153.498
C01285=1084.612,139.543,-68.392,174.979,21.356,153.498
C01286=1084.606,139.294,-68.372,174.978,21.354,153.498
C01287=1084.600,139.045,-68.352,174.976,21.352,153.498
C01288=1084.594,138.796,-68.332,174.973,21.350,153.498
C01289=1084.589,138.547,-68.311,174.971,21.349,153.498
C01290=1084.583,138.298,-68.292,174.969,21.347,153.498
C01291=1084.578,138.049,-68.271,174.967,21.345,153.498
C01292=1084.572,137.800,-68.251,174.965,21.343,153.498
C01293=1084.567,137.551,-68.231,174.963,21.341,153.498
C01294=1084.561,137.302,-68.211,174.961,21.340,153.498
C01295=1084.556,137.053,-68.190,174.958,21.338,153.498
C01296=1084.550,136.803,-68.171,174.957,21.336,153.498
C01297=1084.545,136.554,-68.150,174.954,21.334,153.498
C01298=1084.539,136.305,-68.131,174.952,21.332,153.498
C01299=1084.533,136.056,-68.110,174.950,21.330,153.498
C01300=1084.527,135.806,-68.090,174.948,21.329,153.498
C01301=1084.521,135.557,-68.070,174.946,21.327,153.498
C01302=1084.516,135.308,-68.050,174.943,21.325,153.498
C01303=1084.510,135.059,-68.030,174.942,21.323,153.497
C01304=1084.505,134.810,-68.010,174.939,21.321,153.497
C01305=1084.499,134.561,-67.990,174.937,21.319,153.497
C01306=1084.494,134.312,-67.970,174.936,21.318,153.497
C01307=1084.488,134.062,-67.950,174.933,21.316,153.497
C01308=1084.482,133.813,-67.930,174.931,21.313,153.497
C01309=1084.477,133.564,-67.910,174.929,21.312,153.497
C01310=1084.471,133.315,-67.891,174.927,21.310,153.497
C01311=1084.466,133.066,-67.870,174.925,21.308,153.497
C01312=1084.460,132.817,-67.850,174.922,21.306,153.497
C01313=1084.454,132.568,-67.831,174.921,21.304,153.497
C01314=1084.449,132.318,-67.810,174.918,21.303,153.497
C01315=1084.443,132.069,-67.791,174.916,21.301,153.497
C01316=1084.437,131.820,-67.771,174.914,21.299,153.497
C01317=1084.431,131.571,-67.751,174.912,21.297,153.497
C01318=1084.426,131.322,-67.731,174.910,21.295,153.497
C01319=1084.420,131.073,-67.711,174.908,21.294,153.497
C01320=1084.415,130.823,-67.692,174.906,21.292,153.497
C01321=1084.409,130.575,-67.672,174.903,21.290,153.497
C01322=1084.403,130.325,-67.653,174.902,21.288,153.497
C01323=1084.398,130.076,-67.632,174.900,21.286,153.497
C01324=1084.392,129.827,-67.613,174.897,21.284,153.496
C01325=1084.386,129.578,-67.593,174.896,21.283,153.496
C01326=1084.380,129.329,-67.573,174.893,21.281,153.496
C01327=1084.374,129.080,-67.554,174.891,21.279,153.496
C01328=1084.369,128.830,-67.535,174.889,21.277,153.496
C01329=1084.363,128.581,-67.514,174.887,21.276,153.496
C01330=1084.358,128.332,-67.495,174.885,21.273,153.496
C01331=1084.352,128.083,-67.475,174.883,21.272,153.496
C01332=1084.345,127.804,-67.454,174.881,21.270,153.496
C01333=1084.339,127.524,-67.431,174.879,21.267,153.496
C01334=1084.333,127.246,-67.410,174.876,21.266,153.496
C01335=1084.326,126.966,-67.387,174.874,21.264,153.496
C01336=1084.321,126.717,-67.368,174.872,21.261,153.496
C01337=1084.315,126.468,-67.348,174.870,21.260,153.496
C01338=1084.310,126.219,-67.329,174.868,21.258,153.496
C01339=1084.304,125.970,-67.309,174.865,21.256,153.496
C01340=1084.298,125.721,-67.290,174.864,21.254,153.496
C01341=1084.293,125.471,-67.270,174.862,21.252,153.496
C01342=1084.287,125.222,-67.250,174.859,21.250,153.496
C01343=1084.281,124.973,-67.231,174.858,21.248,153.495
C01344=1084.276,124.724,-67.212,174.855,21.247,153.495
C01345=1084.270,124.475,-67.192,174.853,21.245,153.495
C01346=1084.264,124.225,-67.172,174.852,21.243,153.495
C01347=1084.259,123.977,-67.153,174.849,21.241,153.495
C01348=1084.253,123.728,-67.133,174.848,21.239,153.495
C01349=1084.247,123.478,-67.114,174.846,21.237,153.495
C01350=1084.241,123.229,-67.095,174.843,21.235,153.495
C01351=1084.236,122.980,-67.076,174.842,21.234,153.495
C01352=1084.230,122.731,-67.056,174.839,21.231,153.495
C01353=1084.225,122.482,-67.036,174.837,21.229,153.495
C01354=1084.220,122.232,-67.017,174.835,21.228,153.495
C01355=1084.214,121.983,-66.998,174.833,21.226,153.495
C01356=1084.208,121.734,-66.978,174.831,21.224,153.495
C01357=1084.202,121.485,-66.959,174.829,21.222,153.495
C01358=1084.197,121.235,-66.939,174.827,21.220,153.494
C01359=1084.192,120.986,-66.921,174.826,21.218,153.494
C01360=1084.186,120.737,-66.901,174.823,21.217,153.494
C01361=1084.180,120.488,-66.882,174.821,21.214,153.494
C01362=1084.174,120.239,-66.862,174.819,21.213,153.494
C01363=1084.168,119.989,-66.843,174.817,21.210,153.494
C01364=1084.163,119.741,-66.824,174.815,21.208,153.494
C01365=1084.158,119.491,-66.805,174.813,21.207,153.494
C01366=1084.152,119.242,-66.785,174.811,21.205,153.494
C01367=1084.146,118.992,-66.766,174.810,21.203,153.494
C01368=1084.141,118.744,-66.747,174.807,21.201,153.494
C01369=1084.135,118.495,-66.727,174.805,21.199,153.494
C01370=1084.130,118.245,-66.708,174.804,21.197,153.493
C01371=1084.124,117.996,-66.689,174.801,21.195,153.493
C01372=1084.119,117.747,-66.670,174.800,21.193,153.493
C01373=1084.113,117.498,-66.651,174.797,21.191,153.493
C01374=1084.107,117.248,-66.632,174.795,21.189,153.493
C01375=1084.102,117.000,-66.613,174.794,21.187,153.493
C01376=1084.097,116.750,-66.593,174.792,21.185,153.493
C01377=1084.091,116.501,-66.574,174.790,21.184,153.493
C01378=1084.085,116.251,-66.555,174.788,21.181,153.493
C01379=1084.080,116.002,-66.536,174.785,21.179,153.493
C01380=1084.074,115.753,-66.517,174.784,21.177,153.493
C01381=1084.069,115.504,-66.498,174.782,21.175,153.493
C01382=1084.064,115.255,-66.479,174.780,21.174,153.492
C01383=1084.058,115.005,-66.459,174.778,21.172,153.492
C01384=1084.052,114.756,-66.440,174.776,21.169,153.492
C01385=1084.047,114.507,-66.421,174.774,21.168,153.492
C01386=1084.041,114.258,-66.403,174.772,21.165,153.492
C01387=1084.035,114.009,-66.383,174.770,21.164,153.492
C01388=1084.029,113.759,-66.364,174.768,21.162,153.492
C01389=1084.024,113.511,-66.345,174.766,21.160,153.492
C01390=1084.019,113.261,-66.327,174.764,21.158,153.492
C01391=1084.013,113.011,-66.308,174.762,21.156,153.492
C01392=1084.007,112.763,-66.289,174.761,21.154,153.492
C01393=1084.002,112.513,-66.270,174.758,21.152,153.491
C01394=1083.996,112.264,-66.251,174.756,21.150,153.491
C01395=1083.990,112.015,-66.232,174.755,21.148,153.491
C01396=1083.983,111.736,-66.211,174.752,21.146,153.491
C01397=1083.978,111.457,-66.189,174.750,21.144,153.491
C01398=1083.971,111.177,-66.170,174.748,21.141,153.491
C01399=1083.965,110.898,-66.148,174.746,21.140,153.491
C01400=1083.959,110.649,-66.129,174.744,21.138,153.491
C01401=1083.954,110.400,-66.110,174.742,21.136,153.491
C01402=1083.948,110.151,-66.092,174.740,21.134,153.491
C01403=1083.942,109.902,-66.072,174.738,21.132,153.491
C01404=1083.937,109.652,-66.054,174.736,21.129,153.490
C01405=1083.930,109.402,-66.035,174.734,21.128,153.490
C01406=1083.925,109.154,-66.016,174.732,21.126,153.490
C01407=1083.920,108.904,-65.997,174.731,21.124,153.490
C01408=1083.913,108.655,-65.979,174.728,21.122,153.490
C01409=1083.908,108.406,-65.960,174.727,21.120,153.490
C01410=1083.902,108.157,-65.942,174.725,21.118,153.490
C01411=1083.897,107.907,-65.924,174.722,21.116,153.490
C01412=1083.891,107.658,-65.904,174.721,21.114,153.490
C01413=1083.885,107.409,-65.886,174.719,21.112,153.490
C01414=1083.880,107.160,-65.867,174.717,21.110,153.490
C01415=1083.874,106.910,-65.849,174.715,21.108,153.490
C01416=1083.868,106.661,-65.830,174.714,21.106,153.489
C01417=1083.863,106.412,-65.811,174.711,21.105,153.489
C01418=1083.857,106.162,-65.793,174.710,21.103,153.489
C01419=1083.852,105.914,-65.774,174.707,21.101,153.489
C01420=1083.846,105.664,-65.756,174.705,21.098,153.489
C01421=1083.840,105.415,-65.737,174.704,21.096,153.489
C01422=1083.835,105.166,-65.718,174.701,21.094,153.489
C01423=1083.829,104.916,-65.700,174.700,21.093,153.489
C01424=1083.824,104.667,-65.681,174.698,21.091,153.489
C01425=1083.817,104.418,-65.662,174.696,21.089,153.488
C01426=1083.812,104.169,-65.644,174.694,21.086,153.488
C01427=1083.806,103.920,-65.626,174.693,21.085,153.488
C01428=1083.801,103.670,-65.607,174.691,21.082,153.488
C01429=1083.795,103.421,-65.589,174.688,21.081,153.488
C01430=1083.789,103.171,-65.570,174.687,21.079,153.488
C01431=1083.784,102.922,-65.551,174.685,21.076,153.488
C01432=1083.778,102.673,-65.533,174.683,21.075,153.488
C01433=1083.773,102.424,-65.515,174.681,21.072,153.488
C01434=1083.767,102.174,-65.497,174.679,21.071,153.488
C01435=1083.762,101.926,-65.478,174.677,21.068,153.487
C01436=1083.756,101.676,-65.460,174.676,21.067,153.487
C01437=1083.751,101.427,-65.441,174.673,21.065,153.487
C01438=1083.745,101.177,-65.423,174.672,21.063,153.487
C01439=1083.740,100.929,-65.404,174.670,21.060,153.487
C01440=1083.733,100.679,-65.386,174.668,21.059,153.487
C01441=1083.728,100.430,-65.368,174.666,21.056,153.487
C01442=1083.722,100.180,-65.349,174.664,21.055,153.487
C01443=1083.716,99.931,-65.331,174.663,21.053,153.487
C01444=1083.710,99.682,-65.313,174.660,21.050,153.486
C01445=1083.705,99.432,-65.295,174.659,21.049,153.486
C01446=1083.699,99.184,-65.276,174.657,21.046,153.486
C01447=1083.693,98.934,-65.258,174.655,21.045,153.486
C01448=1083.688,98.685,-65.240,174.653,21.042,153.486
C01449=1083.682,98.436,-65.222,174.652,21.041,153.486
C01450=1083.676,98.186,-65.204,174.649,21.039,153.486
C01451=1083.671,97.937,-65.185,174.648,21.037,153.486
C01452=1083.665,97.688,-65.167,174.645,21.035,153.486
C01453=1083.659,97.438,-65.149,174.644,21.033,153.485
C01454=1083.654,97.190,-65.130,174.642,21.030,153.485
C01455=1083.648,96.940,-65.112,174.640,21.029,153.485
C01456=1083.642,96.691,-65.095,174.638,21.027,153.485
C01457=1083.636,96.441,-65.076,174.637,21.025,153.485
C01458=1083.631,96.192,-65.058,174.635,21.023,153.485
C01459=1083.625,95.943,-65.040,174.633,21.021,153.485
C01460=1083.619,95.664,-65.019,174.631,21.018,153.485
C01461=1083.613,95.385,-65.000,174.629,21.016,153.485
C01462=1083.607,95.106,-64.979,174.627,21.014,153.484
C01463=1083.600,94.826,-64.959,174.624,21.011,153.484
C01464=1083.593,94.577,-64.941,174.623,21.010,153.484
C01465=1083.589,94.328,-64.923,174.621,21.007,153.484
C01466=1083.583,94.079,-64.905,174.619,21.005,153.484
C01467=1083.577,93.829,-64.887,174.617,21.003,153.484
C01468=1083.572,93.580,-64.870,174.616,21.001,153.484
C01469=1083.566,93.331,-64.850,174.614,20.999,153.484
C01470=1083.560,93.082,-64.833,174.612,20.997,153.483
C01471=1083.555,92.833,-64.815,174.610,20.995,153.483
C01472=1083.549,92.583,-64.797,174.608,20.993,153.483
C01473=1083.544,92.333,-64.779,174.606,20.991,153.483
C01474=1083.538,92.084,-64.760,174.605,20.989,153.483
C01475=1083.532,91.835,-64.743,174.603,20.987,153.483
C01476=1083.526,91.586,-64.725,174.601,20.985,153.483
C01477=1083.521,91.336,-64.707,174.599,20.983,153.483
C01478=1083.516,91.087,-64.689,174.598,20.981,153.482
C01479=1083.510,90.838,-64.672,174.595,20.979,153.482
C01480=1083.504,90.588,-64.654,174.594,20.977,153.482
C01481=1083.498,90.339,-64.636,174.592,20.974,153.482
C01482=1083.492,90.090,-64.618,174.591,20.972,153.482
C01483=1083.487,89.841,-64.601,174.588,20.970,153.482
C01484=1083.480,89.591,-64.582,174.587,20.969,153.482
C01485=1083.475,89.342,-64.564,174.585,20.966,153.482
C01486=1083.469,89.093,-64.547,174.583,20.965,153.482
C01487=1083.463,88.844,-64.529,174.581,20.962,153.481
C01488=1083.458,88.595,-64.511,174.580,20.960,153.481
C01489=1083.452,88.344,-64.493,174.577,20.958,153.481
C01490=1083.447,88.095,-64.475,174.576,20.956,153.481
C01491=1083.441,87.846,-64.458,174.574,20.954,153.481
C01492=1083.435,87.597,-64.440,174.572,20.952,153.481
C01493=1083.430,87.348,-64.422,174.570,20.950,153.481
C01494=1083.424,87.099,-64.405,174.569,20.948,153.481
C01495=1083.418,86.849,-64.387,174.567,20.946,153.480
C01496=1083.412,86.600,-64.369,174.565,20.944,153.480
C01497=1083.407,86.351,-64.352,174.563,20.942,153.480
C01498=1083.401,86.101,-64.334,174.562,20.940,153.480
C01499=1083.395,85.852,-64.316,174.559,20.938,153.480
C01500=1083.390,85.602,-64.299,174.558,20.936,153.480
C01501=1083.384,85.353,-64.281,174.557,20.934,153.480
C01502=1083.378,85.104,-64.264,174.554,20.932,153.480
C01503=1083.373,84.855,-64.246,174.553,20.930,153.479
C01504=1083.367,84.605,-64.228,174.551,20.927,153.479
C01505=1083.361,84.356,-64.211,174.550,20.925,153.479
C01506=1083.356,84.107,-64.193,174.547,20.923,153.479
C01507=1083.349,83.857,-64.176,174.546,20.922,153.479
C01508=1083.343,83.608,-64.158,174.544,20.919,153.479
C01509=1083.338,83.359,-64.141,174.542,20.917,153.479
C01510=1083.333,83.110,-64.124,174.540,20.915,153.478
C01511=1083.327,82.860,-64.106,174.539,20.913,153.478
C01512=1083.321,82.611,-64.088,174.536,20.911,153.478
C01513=1083.315,82.362,-64.071,174.535,20.909,153.478
C01514=1083.310,82.112,-64.054,174.533,20.906,153.478
C01515=1083.304,81.862,-64.036,174.532,20.905,153.478
C01516=1083.299,81.613,-64.018,174.529,20.902,153.478
C01517=1083.293,81.364,-64.001,174.528,20.900,153.477
C01518=1083.288,81.115,-63.983,174.527,20.898,153.477
C01519=1083.282,80.865,-63.966,174.524,20.896,153.477
C01520=1083.276,80.616,-63.948,174.523,20.894,153.477
C01521=1083.271,80.367,-63.931,174.521,20.892,153.477
C01522=1083.265,80.118,-63.913,174.520,20.890,153.477
C01523=1083.259,79.867,-63.896,174.517,20.888,153.477
C01524=1083.253,79.589,-63.877,174.515,20.885,153.476
C01525=1083.247,79.310,-63.857,174.514,20.883,153.476
C01526=1083.241,79.031,-63.837,174.512,20.881,153.476
C01527=1083.234,78.751,-63.818,174.510,20.878,153.476
C01528=1083.228,78.502,-63.801,174.508,20.876,153.476
C01529=1083.222,78.253,-63.784,174.506,20.874,153.476
C01530=1083.217,78.004,-63.767,174.505,20.872,153.476
C01531=1083.211,77.754,-63.749,174.503,20.870,153.475
C01532=1083.206,77.505,-63.732,174.501,20.868,153.475
C01533=1083.200,77.256,-63.715,174.500,20.866,153.475
C01534=1083.194,77.007,-63.698,174.498,20.864,153.475
C01535=1083.189,76.758,-63.680,174.496,20.862,153.475
C01536=1083.182,76.508,-63.663,174.494,20.859,153.475
C01537=1083.177,76.258,-63.646,174.493,20.857,153.475
C01538=1083.171,76.009,-63.629,174.491,20.855,153.474
C01539=1083.166,75.760,-63.612,174.489,20.853,153.474
C01540=1083.160,75.511,-63.595,174.487,20.851,153.474
C01541=1083.154,75.261,-63.577,174.486,20.849,153.474
C01542=1083.148,75.012,-63.560,174.484,20.847,153.474
C01543=1083.142,74.762,-63.543,174.482,20.845,153.474
C01544=1083.137,74.513,-63.526,174.481,20.843,153.474
C01545=1083.132,74.264,-63.509,174.479,20.840,153.473
C01546=1083.125,74.014,-63.492,174.477,20.838,153.473
C01547=1083.119,73.765,-63.475,174.475,20.836,153.473
C01548=1083.114,73.515,-63.457,174.474,20.834,153.473
C01549=1083.109,73.266,-63.440,174.472,20.832,153.473
C01550=1083.102,73.017,-63.423,174.470,20.830,153.473
C01551=1083.097,72.767,-63.407,174.469,20.828,153.472
C01552=1083.092,72.518,-63.389,174.467,20.825,153.472
C01553=1083.085,72.268,-63.372,174.465,20.824,153.472
C01554=1083.080,72.019,-63.355,174.463,20.821,153.472
C01555=1083.074,71.770,-63.339,174.462,20.819,153.472
C01556=1083.068,71.521,-63.321,174.460,20.817,153.472
C01557=1083.063,71.271,-63.304,174.458,20.815,153.472
C01558=1083.057,71.023,-63.287,174.457,20.813,153.471
C01559=1083.052,70.773,-63.270,174.455,20.811,153.471
C01560=1083.046,70.523,-63.254,174.454,20.809,153.471
C01561=1083.040,70.274,-63.237,174.452,20.806,153.471
C01562=1083.034,70.024,-63.219,174.450,20.804,153.471
C01563=1083.028,69.775,-63.202,174.448,20.802,153.471
C01564=1083.023,69.526,-63.186,174.447,20.800,153.471
C01565=1083.017,69.276,-63.169,174.445,20.798,153.470
C01566=1083.011,69.027,-63.152,174.443,20.795,153.470
C01567=1083.006,68.778,-63.135,174.442,20.793,153.470
C01568=1083.000,68.528,-63.119,174.440,20.791,153.470
C01569=1082.995,68.279,-63.101,174.438,20.790,153.470
C01570=1082.989,68.030,-63.085,174.437,20.788,153.470
C01571=1082.983,67.780,-63.068,174.435,20.785,153.470
C01572=1082.977,67.531,-63.051,174.433,20.783,153.469
C01573=1082.971,67.281,-63.034,174.431,20.781,153.469
C01574=1082.965,67.032,-63.017,174.430,20.779,153.469
C01575=1082.960,66.783,-63.000,174.428,20.776,153.469
C01576=1082.954,66.533,-62.984,174.427,20.774,153.469
C01577=1082.949,66.284,-62.967,174.425,20.772,153.469
C01578=1082.943,66.034,-62.951,174.423,20.770,153.468
C01579=1082.937,65.786,-62.934,174.422,20.768,153.468
C01580=1082.931,65.536,-62.917,174.420,20.766,153.468
C01581=1082.925,65.287,-62.900,174.418,20.764,153.468
C01582=1082.920,65.037,-62.884,174.417,20.762,153.468
C01583=1082.914,64.788,-62.867,174.415,20.759,153.468
C01584=1082.909,64.539,-62.850,174.413,20.757,153.467
C01585=1082.903,64.289,-62.834,174.411,20.755,153.467
C01586=1082.897,64.040,-62.817,174.410,20.753,153.467
C01587=1082.891,63.790,-62.800,174.409,20.751,153.467
C01588=1082.884,63.511,-62.781,174.407,20.748,153.467
C01589=1082.878,63.233,-62.763,174.404,20.746,153.467
C01590=1082.871,62.953,-62.744,174.402,20.744,153.467
C01591=1082.865,62.674,-62.726,174.401,20.742,153.466
C01592=1082.859,62.425,-62.710,174.399,20.739,153.466
C01593=1082.853,62.175,-62.693,174.397,20.737,153.466
C01594=1082.848,61.926,-62.677,174.396,20.735,153.466
C01595=1082.842,61.676,-62.660,174.394,20.733,153.466
C01596=1082.835,61.427,-62.643,174.393,20.731,153.466
C01597=1082.829,61.177,-62.627,174.391,20.728,153.465
C01598=1082.824,60.928,-62.610,174.389,20.726,153.465
C01599=1082.818,60.678,-62.594,174.388,20.724,153.465
C01600=1082.812,60.429,-62.577,174.386,20.722,153.465
C01601=1082.806,60.180,-62.561,174.384,20.720,153.465
C01602=1082.800,59.930,-62.545,174.382,20.718,153.465
C01603=1082.795,59.681,-62.528,174.381,20.716,153.465
C01604=1082.789,59.431,-62.512,174.379,20.714,153.464
C01605=1082.783,59.182,-62.495,174.377,20.712,153.464
C01606=1082.777,58.933,-62.479,174.376,20.710,153.464
C01607=1082.772,58.683,-62.462,174.375,20.708,153.464
C01608=1082.766,58.434,-62.446,174.373,20.705,153.464
C01609=1082.760,58.184,-62.430,174.371,20.703,153.464
C01610=1082.754,57.935,-62.414,174.369,20.701,153.463
C01611=1082.748,57.686,-62.397,174.368,20.699,153.463
C01612=1082.743,57.436,-62.380,174.366,20.697,153.463
C01613=1082.737,57.187,-62.364,174.364,20.695,153.463
C01614=1082.731,56.937,-62.348,174.363,20.693,153.463
C01615=1082.725,56.689,-62.332,174.361,20.690,153.463
C01616=1082.719,56.439,-62.316,174.360,20.688,153.462
C01617=1082.713,56.190,-62.300,174.358,20.686,153.462
C01618=1082.708,55.940,-62.283,174.356,20.684,153.462
C01619=1082.702,55.691,-62.266,174.355,20.682,153.462
C01620=1082.696,55.442,-62.250,174.353,20.680,153.462
C01621=1082.690,55.192,-62.234,174.351,20.677,153.462
C01622=1082.684,54.943,-62.218,174.350,20.675,153.461
C01623=1082.679,54.693,-62.202,174.348,20.673,153.461
C01624=1082.674,54.443,-62.185,174.347,20.671,153.461
C01625=1082.668,54.194,-62.169,174.345,20.669,153.461
C01626=1082.662,53.944,-62.153,174.343,20.666,153.461
C01627=1082.656,53.695,-62.137,174.342,20.664,153.461
C01628=1082.650,53.446,-62.121,174.341,20.662,153.460
C01629=1082.644,53.197,-62.104,174.339,20.660,153.460
C01630=1082.639,52.947,-62.089,174.337,20.658,153.460
C01631=1082.633,52.698,-62.073,174.335,20.655,153.460
C01632=1082.628,52.448,-62.056,174.334,20.653,153.460
C01633=1082.622,52.199,-62.039,174.332,20.651,153.460
C01634=1082.616,51.949,-62.023,174.330,20.649,153.459
C01635=1082.610,51.700,-62.007,174.329,20.647,153.459
C01636=1082.605,51.451,-61.992,174.328,20.645,153.459
C01637=1082.599,51.202,-61.976,174.326,20.642,153.459
C01638=1082.593,50.952,-61.959,174.324,20.640,153.459
C01639=1082.587,50.703,-61.943,174.322,20.638,153.459
C01640=1082.581,50.453,-61.927,174.321,20.636,153.458
C01641=1082.576,50.203,-61.911,174.320,20.634,153.458
C01642=1082.571,49.955,-61.895,174.318,20.631,153.458
C01643=1082.565,49.705,-61.878,174.316,20.629,153.458
C01644=1082.559,49.455,-61.863,174.315,20.627,153.458
C01645=1082.553,49.206,-61.847,174.313,20.625,153.458
C01646=1082.547,48.957,-61.830,174.312,20.622,153.457
C01647=1082.542,48.707,-61.815,174.310,20.620,153.457
C01648=1082.536,48.458,-61.799,174.308,20.618,153.457
C01649=1082.530,48.209,-61.783,174.307,20.616,153.457
C01650=1082.525,47.959,-61.767,174.305,20.614,153.457
C01651=1082.519,47.709,-61.751,174.304,20.612,153.456
C01652=1082.513,47.429,-61.733,174.302,20.609,153.456
C01653=1082.507,47.151,-61.715,174.300,20.607,153.456
C01654=1082.500,46.871,-61.697,174.298,20.604,153.456
C01655=1082.494,46.592,-61.679,174.297,20.602,153.456
C01656=1082.488,46.342,-61.664,174.295,20.599,153.455
C01657=1082.482,46.093,-61.648,174.294,20.597,153.455
C01658=1082.476,45.844,-61.631,174.291,20.595,153.455
C01659=1082.471,45.594,-61.616,174.290,20.592,153.455
C01660=1082.465,45.345,-61.600,174.289,20.590,153.455
C01661=1082.460,45.095,-61.584,174.287,20.588,153.454
C01662=1082.454,44.846,-61.568,174.286,20.586,153.454
C01663=1082.449,44.596,-61.553,174.284,20.584,153.454
C01664=1082.443,44.347,-61.537,174.282,20.581,153.454
C01665=1082.437,44.098,-61.520,174.281,20.579,153.454
C01666=1082.432,43.849,-61.505,174.280,20.577,153.454
C01667=1082.426,43.599,-61.489,174.278,20.575,153.453
C01668=1082.420,43.349,-61.473,174.276,20.573,153.453
C01669=1082.414,43.100,-61.457,174.275,20.571,153.453
C01670=1082.409,42.850,-61.442,174.273,20.568,153.453
C01671=1082.403,42.601,-61.426,174.272,20.566,153.453
C01672=1082.397,42.352,-61.411,174.270,20.564,153.453
C01673=1082.391,42.102,-61.395,174.268,20.561,153.452
C01674=1082.385,41.852,-61.379,174.267,20.559,153.452
C01675=1082.380,41.604,-61.363,174.266,20.557,153.452
C01676=1082.374,41.354,-61.348,174.264,20.555,153.452
C01677=1082.369,41.104,-61.332,174.262,20.553,153.452
C01678=1082.363,40.855,-61.317,174.261,20.551,153.451
C01679=1082.357,40.605,-61.301,174.259,20.548,153.451
C01680=1082.351,40.356,-61.285,174.258,20.546,153.451
C01681=1082.345,40.106,-61.269,174.257,20.544,153.451
C01682=1082.340,39.857,-61.253,174.254,20.542,153.451
C01683=1082.334,39.608,-61.239,174.253,20.540,153.451
C01684=1082.328,39.358,-61.223,174.252,20.538,153.450
C01685=1082.323,39.109,-61.207,174.250,20.535,153.450
C01686=1082.317,38.859,-61.192,174.248,20.533,153.450
C01687=1082.311,38.610,-61.175,174.247,20.531,153.450
C01688=1082.305,38.361,-61.161,174.245,20.528,153.450
C01689=1082.300,38.111,-61.145,174.244,20.526,153.449
C01690=1082.294,37.862,-61.129,174.243,20.524,153.449
C01691=1082.289,37.612,-61.114,174.240,20.522,153.449
C01692=1082.282,37.363,-61.099,174.239,20.520,153.449
C01693=1082.276,37.113,-61.083,174.238,20.518,153.449
C01694=1082.271,36.863,-61.067,174.236,20.515,153.449
C01695=1082.265,36.614,-61.052,174.234,20.513,153.448
C01696=1082.259,36.364,-61.037,174.233,20.511,153.448
C01697=1082.252,36.115,-61.021,174.231,20.508,153.448
C01698=1082.247,35.866,-61.006,174.230,20.506,153.448
C01699=1082.242,35.616,-60.991,174.229,20.504,153.448
C01700=1082.235,35.367,-60.975,174.226,20.502,153.448
C01701=1082.230,35.118,-60.960,174.225,20.500,153.447
C01702=1082.224,34.868,-60.944,174.224,20.498,153.447
C01703=1082.218,34.618,-60.929,174.222,20.496,153.447
C01704=1082.213,34.370,-60.913,174.220,20.494,153.447
C01705=1082.206,34.120,-60.898,174.219,20.491,153.447
C01706=1082.201,33.870,-60.883,174.217,20.489,153.446
C01707=1082.196,33.621,-60.868,174.216,20.487,153.446
C01708=1082.189,33.371,-60.853,174.215,20.485,153.446
C01709=1082.183,33.122,-60.836,174.212,20.482,153.446
C01710=1082.177,32.873,-60.822,174.211,20.480,153.446
C01711=1082.172,32.623,-60.806,174.210,20.478,153.446
C01712=1082.167,32.373,-60.791,174.208,20.475,153.445
C01713=1082.160,32.124,-60.776,174.207,20.473,153.445
C01714=1082.154,31.874,-60.760,174.205,20.471,153.445
C01715=1082.149,31.625,-60.745,174.204,20.469,153.445
C01716=1082.142,31.346,-60.728,174.202,20.467,153.445
C01717=1082.136,31.066,-60.712,174.200,20.464,153.444
C01718=1082.130,30.787,-60.694,174.199,20.462,153.444
C01719=1082.123,30.507,-60.677,174.197,20.459,153.444
C01720=1082.117,30.258,-60.662,174.195,20.457,153.444
C01721=1082.112,30.008,-60.647,174.194,20.455,153.444
C01722=1082.105,29.759,-60.631,174.192,20.453,153.443
C01723=1082.100,29.510,-60.616,174.191,20.451,153.443
C01724=1082.094,29.260,-60.601,174.190,20.448,153.443
C01725=1082.088,29.010,-60.586,174.188,20.446,153.443
C01726=1082.082,28.762,-60.571,174.186,20.444,153.443
C01727=1082.077,28.512,-60.556,174.185,20.442,153.442
C01728=1082.071,28.263,-60.541,174.183,20.439,153.442
C01729=1082.065,28.013,-60.525,174.182,20.437,153.442
C01730=1082.060,27.764,-60.511,174.180,20.435,153.442
C01731=1082.054,27.514,-60.495,174.178,20.433,153.442
C01732=1082.048,27.264,-60.480,174.177,20.430,153.442
C01733=1082.042,27.015,-60.466,174.176,20.428,153.441
C01734=1082.036,26.765,-60.450,174.174,20.426,153.441
C01735=1082.030,26.516,-60.436,174.172,20.424,153.441
C01736=1082.025,26.266,-60.420,174.171,20.422,153.441
C01737=1082.019,26.017,-60.405,174.170,20.420,153.441
C01738=1082.013,25.768,-60.391,174.168,20.417,153.441
C01739=1082.007,25.518,-60.375,174.167,20.415,153.440
C01740=1082.001,25.269,-60.360,174.165,20.413,153.440
C01741=1081.995,25.019,-60.345,174.164,20.411,153.440
C01742=1081.990,24.770,-60.330,174.162,20.408,153.440
C01743=1081.983,24.520,-60.315,174.161,20.406,153.440
C01744=1081.978,24.271,-60.300,174.159,20.405,153.439
C01745=1081.972,24.021,-60.286,174.157,20.402,153.439
C01746=1081.966,23.772,-60.271,174.156,20.400,153.439
C01747=1081.961,23.522,-60.256,174.155,20.398,153.439
C01748=1081.955,23.273,-60.241,174.153,20.395,153.439
C01749=1081.949,23.023,-60.226,174.151,20.393,153.439
C01750=1081.944,22.774,-60.211,174.150,20.391,153.438
C01751=1081.937,22.524,-60.196,174.149,20.389,153.438
C01752=1081.931,22.275,-60.182,174.147,20.387,153.438
C01753=1081.926,22.025,-60.167,174.146,20.384,153.438
C01754=1081.920,21.776,-60.152,174.144,20.382,153.438
C01755=1081.914,21.526,-60.137,174.142,20.380,153.437
C01756=1081.909,21.277,-60.122,174.141,20.378,153.437
C01757=1081.902,21.027,-60.107,174.140,20.376,153.437
C01758=1081.897,20.778,-60.093,174.138,20.374,153.437
C01759=1081.891,20.528,-60.078,174.136,20.371,153.437
C01760=1081.886,20.279,-60.063,174.135,20.369,153.436
C01761=1081.879,20.029,-60.048,174.134,20.367,153.436
C01762=1081.873,19.780,-60.034,174.132,20.364,153.436
C01763=1081.868,19.531,-60.019,174.130,20.362,153.436
C01764=1081.862,19.280,-60.004,174.129,20.360,153.436
C01765=1081.856,19.031,-59.990,174.128,20.358,153.436
C01766=1081.850,18.782,-59.975,174.126,20.356,153.436
C01767=1081.844,18.533,-59.960,174.125,20.353,153.435
C01768=1081.838,18.283,-59.946,174.123,20.351,153.435
C01769=1081.833,18.033,-59.931,174.122,20.349,153.435
C01770=1081.827,17.784,-59.916,174.120,20.347,153.435
C01771=1081.821,17.534,-59.902,174.119,20.345,153.435
C01772=1081.815,17.284,-59.887,174.117,20.343,153.434
C01773=1081.809,17.035,-59.872,174.115,20.341,153.434
C01774=1081.804,16.786,-59.857,174.114,20.338,153.434
C01775=1081.798,16.536,-59.843,174.113,20.336,153.434
C01776=1081.792,16.287,-59.828,174.112,20.334,153.434
C01777=1081.786,16.037,-59.813,174.109,20.332,153.433
C01778=1081.780,15.788,-59.800,174.108,20.330,153.433
C01779=1081.774,15.538,-59.785,174.107,20.328,153.433
C01780=1081.768,15.239,-59.768,174.105,20.325,153.433
C01781=1081.761,14.939,-59.750,174.103,20.322,153.433
C01782=1081.754,14.639,-59.732,174.102,20.320,153.432
C01783=1081.747,14.339,-59.715,174.100,20.317,153.432
C01784=1081.741,14.090,-59.700,174.099,20.315,153.432
C01785=1081.735,13.841,-59.685,174.096,20.312,153.432
C01786=1081.729,13.591,-59.672,174.095,20.310,153.432
C01787=1081.723,13.341,-59.657,174.094,20.308,153.431
C01788=1081.717,13.092,-59.643,174.093,20.306,153.431
C01789=1081.712,12.843,-59.628,174.090,20.304,153.431
C01790=1081.706,12.593,-59.614,174.089,20.302,153.431
C01791=1081.700,12.344,-59.599,174.088,20.300,153.431
C01792=1081.693,12.094,-59.584,174.087,20.298,153.431
C01793=1081.688,11.844,-59.570,174.084,20.295,153.431
C01794=1081.682,11.595,-59.556,174.083,20.293,153.430
C01795=1081.676,11.345,-59.542,174.082,20.291,153.430
C01796=1081.670,11.096,-59.527,174.080,20.288,153.430
C01797=1081.664,10.846,-59.513,174.079,20.286,153.430
C01798=1081.658,10.597,-59.499,174.077,20.284,153.430
C01799=1081.652,10.348,-59.485,174.076,20.282,153.429
C01800=1081.646,10.098,-59.470,174.074,20.280,153.429
C01801=1081.640,9.849,-59.456,174.073,20.278,153.429
C01802=1081.634,9.599,-59.441,174.071,20.276,153.429
C01803=1081.629,9.349,-59.427,174.070,20.274,153.429
C01804=1081.623,9.100,-59.414,174.068,20.271,153.429
C01805=1081.617,8.850,-59.399,174.067,20.269,153.428
C01806=1081.611,8.600,-59.385,174.066,20.267,153.428
C01807=1081.605,8.352,-59.370,174.064,20.265,153.428
C01808=1081.599,8.101,-59.356,174.062,20.262,153.428
C01809=1081.594,7.852,-59.341,174.061,20.260,153.428
C01810=1081.588,7.603,-59.327,174.060,20.258,153.427
C01811=1081.582,7.352,-59.313,174.058,20.257,153.427
C01812=1081.576,7.103,-59.299,174.056,20.254,153.427
